(* CODESYS project CoreMotionNc2.library
   Version: 1.1.8
   Title: CoreMotionNc2
   DefaultNamespace: CoreMotionNc2
   Placeholder: CoreMotionNc2
   Company: Beckhoff Automation LLC

Project tree, tasks and I/O mapping:
  libraries: Core, * (Beckhoff Automation LLC); Tc2_MC2, * (Beckhoff Automation GmbH); Tc2_MC2_Drive, * (Beckhoff Automation GmbH); Tc2_NcKinematicTransformation, * (Beckhoff Automation GmbH); Tc2_Standard, * (Beckhoff Automation GmbH); Tc2_System, * (Beckhoff Automation GmbH)
  _Internal/
    Interface/
      interface I_AxisRef: Axis
      interface I_MotionJogTask: JogBackwards, JogForward, Mode, Position
      interface I_MotionPowerTask
      interface I_MotionTask: Axis, Name
      interface I_MotionTaskCollection: AddTask, ErrorTask, RemoveTaskByInstance
    MotionTasks/
      AX5000/
        DUT/
          P_0_0074/
            data type ST_IDN_P_0_0074
            data type ST_IDN_P_0_0074_UDINT
          P_0_0074_LREAL/
            data type ST_IDN_P_0_0074_LREAL
          data type ST_AX5000AmpToNm
        function block MotionTask_AX5000AmpToNm [ST]: ActCurrent, ActTorque, Busy, CyclicLogic, Error, ErrorId, Execute
      Base/
        DUT/
          data type ST_TaskState
        function block MotionTask [ST]: Axis, Busy, CyclicLogic, Error, ErrorId, Execute, Name
        function block MotionTaskCollection [ST]: Busy, Error, ErrorId, ErrorTask, AddTask, CyclicLogic, FB_Init, RemoveTaskByInstance, Reset
      Coupling/
        function block MotionCoupleTask_Gearing [ST]: BufferMode, Busy, CyclicLogic, Error, ErrorId, Execute, GearIn, GearInMultiMasterOptions, GearRatioMaster1, GearRatioMaster2, GearRatioMaster3, GearRatioMaster4, Master1, Master2, Master3, Master4
      Home/
        function block MotionHomeTask_CoESetEncoderOffset [ST]: Busy, CyclicLogic, Error, ErrorId, Execute, HomePosition
        function block MotionHomeTask_SetPosition [ST]: Busy, CyclicLogic, Error, ErrorId, Execute, HomePosition
        function block MotionHomeTask_SetPositionOffset [ST]: Busy, CyclicLogic, Error, ErrorId, Execute, Feedback, HomePosition, Memory
        function block MotionHomeTask_SetZeroHere [ST]: Busy, CyclicLogic, Error, ErrorId, Execute
      Move/
        function block MoveAbsoluteTask [ST]: BufferMode, Busy, CyclicLogic, Error, ErrorId, Execute, MoveOptions, TargetPosition
        function block MoveJogTask [ST]: Busy, CyclicLogic, Error, ErrorId, Execute, JogBackwards, JogForward, Mode, Position
        function block MoveModuloTask [ST]: BufferMode, Busy, CyclicLogic, Direction, Error, ErrorId, Execute, MoveOptions, TargetPosition
        function block MoveRelativeTask [ST]: BufferMode, Busy, CyclicLogic, Error, ErrorId, Execute, MoveOptions, TargetDistance
        function block MoveVelocityTask [ST]: BufferMode, Busy, CyclicLogic, Error, ErrorId, Execute, MoveOptions, TargetVelocity
      Power/
        function block PowerTask [ST]: Busy, CyclicLogic, Disable, Enable, Enabled, Error, ErrorId, Execute, InhibitFeedBackward, InhibitFeedForward, Override
        function block StopTask [ST]: BufferMode, Busy, CyclicLogic, Error, ErrorId, Execute, MoveOptions
      Reset/
        function block CoEExtendedResetTask [ST]: Busy, CyclicLogic, Error, ErrorId, Execute
        function block CoEResetTask [ST]: Busy, CyclicLogic, Error, ErrorId, Execute
        function block SoEResetTask [ST]: Busy, CyclicLogic, Error, ErrorId, Execute
  Kinematic Group/
    Interface/
      interface I_KinematicGroup: AddAcsAxis, AddMcsAxis, BuildGroup, DissolveGroup, Status
    function block KinematicGroup [ST]: DeregisterWithParent, RegisterWithParent, CyclicLogic, Initialize, Initialized, AddAcsAxis, AddMcsAxis, BuildGroup, DissolveGroup, Override, Status, Reset, Busy, Error, ErrorId
    function block KinematicGroup_TcEvents [ST]: GetHighestActiveEventReaction, GetHighestActiveEventSeverity, Reset, SetEventReactions, CyclicLogic, FB_Init
  Motion/
    DUT/
      data type ST_AxisPTP_HMI
      data type ST_MotionDefaults
    Interface/
      interface I_Axis: ErrorId, MotionTasks
      interface I_Axis_PTP
      interface I_AxisDynamics: Acceleration, BufferMode, Deceleration, Jerk, MoveOptions, Velocity
      interface I_AxisEnable: InhibitFeedBackward, InhibitFeedForward
      interface I_AxisGear: GearIn, GearInMultiMasterOptions, GearOut, GearRatioMaster1, GearRatioMaster2, GearRatioMaster3, GearRatioMaster4, Master1, Master2, Master3, Master4
      interface I_AxisHome: Home
      interface I_AxisJog: Jog
      interface I_AxisMoveAbsolute: MoveAbsolute
      interface I_AxisMoveModulo: MoveModulo
      interface I_AxisMoveRelative: MoveRelative
      interface I_AxisMoveVelocity: MoveVelocity
      interface I_AxisStatus: ActualAcceleration, ActualPosition, ActualPositionModulo, ActualTorque, ActualVelocity, AxisParameterSet, Enabled, PositionLag, SetAcceleration, SetPosition, SetPositionModulo, SetVelocity, Stopped
      interface I_SlaveAxis
    function block Axis [ST]: FB_Init, RegisterWithParent, CyclicLogic, Acceleration, BufferMode, Deceleration, Jerk, MoveOptions, Velocity, Disable, Enable, Enabled, InhibitFeedBackward, InhibitFeedForward, Override, Home, HomeTask, Initialize, Initialized, Jog, Reset, ResetTask, ActualAcceleration, ActualPosition, ActualPositionModulo, ActualTorque, ActualVelocity, AxisParameterSet, Busy, Error, ErrorId, PositionLag, SetAcceleration, SetPosition, SetPositionModulo, SetVelocity, Stop, Stopped, StopTask, Axis, MotionTasks
    function block Axis_TcEvents [ST]: GetHighestActiveEventReaction, GetHighestActiveEventSeverity, Reset, SetEventReactions, CyclicLogic, FB_Init
    function block AxisPTP [ST]: FB_Init, MoveAbsolute, MoveModulo, MoveRelative, MoveVelocity
    function block AxisPTP_HMI [ST]: DisablePermissive, EnablePermissive, HomePermissive, JogBackwardFastPermissive, JogBackwardSlowPermissive, JogForwardFastPermissive, JogForwardSlowPermissive, MoveAbsolutePermissive, MoveModuloPermissive, MoveRelativePermissive, MoveVelocityPermissive, ResetPermissive, StopPermissive, ControlObject, CyclicLogic, FB_Init
    function block SlaveAxisPTP [ST]: FB_Init, GearIn, GearInMultiMasterOptions, GearOut, GearRatioMaster1, GearRatioMaster2, GearRatioMaster3, GearRatioMaster4, Master1, Master2, Master3, Master4
  Project Information/
    function F_GetCompany [ST]
    function F_GetTitle [ST]
    function F_GetVersion [ST]
  Version/
    global variables Global_Version
  global variables CoreMotionParameterNc2
*)

// _Internal/MotionTasks/AX5000/DUT/P_0_0074/ST_IDN_P_0_0074
TYPE ST_IDN_P_0_0074 :
	STRUCT
		Iq : ARRAY[0..9] OF UDINT; // Amps ( units := A x 100 )
		M  : ARRAY[0..9] OF UDINT; // Newton Meters ( units := Nm x 100 )
	END_STRUCT
END_TYPE

// _Internal/MotionTasks/AX5000/DUT/P_0_0074/ST_IDN_P_0_0074_UDINT
TYPE ST_IDN_P_0_0074_UDINT :
	STRUCT
		Actual	 : UINT;
		_Max	 : UINT;
		Elements : ST_IDN_P_0_0074;
	END_STRUCT
END_TYPE

// _Internal/MotionTasks/AX5000/DUT/P_0_0074_LREAL/ST_IDN_P_0_0074_LREAL
TYPE ST_IDN_P_0_0074_LREAL :
	STRUCT
		Iq : ARRAY[0..9] OF LREAL;
		M  : ARRAY[0..9] OF LREAL;
	END_STRUCT
END_TYPE

// _Internal/MotionTasks/AX5000/DUT/ST_AX5000AmpToNm
TYPE ST_AX5000AmpToNm :
	STRUCT
		Curve	   : ST_IDN_P_0_0074_LREAL; // Contents read in from P-0-0074   ( scaled )
		ActCurrent : LREAL;					// Actual current in Amps           ( units := A )
		ActTorque  : LREAL;					// Actual torque in Newton Meters   ( units := Nm )
	END_STRUCT
END_TYPE

// _Internal/MotionTasks/Base/DUT/ST_TaskState
TYPE ST_TaskState :
	STRUCT
		Name	: T_MaxString;
		Busy	: BOOL;
		Error	: BOOL;
		ErrorId : UDINT;
	END_STRUCT
END_TYPE

// Motion/DUT/ST_AxisPTP_HMI
TYPE ST_AxisPTP_HMI EXTENDS ST_HmiFunction :
	STRUCT
		Unit				 : STRING;
		Busy				 : BOOL;
		Error				 : BOOL;
		ErrorId				 : UDINT;
		ActualAcceleration	 : LREAL;
		ActualPosition		 : LREAL;
		ActualPositionModulo : LREAL;
		ActualTorque		 : LREAL;
		ActualVelocity		 : LREAL;
		Status				 : ST_AxisStatus;
		Enable				 : Button;
		Disable				 : Button;
		Stop				 : Button;
		JogForwardSlow		 : Button;
		JogBackwardSlow		 : Button;
		JogForwardFast		 : Button;
		JogBackwardFast		 : Button;
		Home				 : Button;
		Reset				 : Button;
		MoveAbsolute		 : Button;
		TargetPosition		 : LREAL;
		MoveVelocity		 : Button;
		TargetVelocity		 : LREAL;
		MoveRelative		 : Button;
		TargetDistance		 : LREAL;
		MoveModulo			 : Button;
	END_STRUCT
END_TYPE

// Motion/DUT/ST_MotionDefaults
TYPE ST_MotionDefaults :
	STRUCT
		DefaultResetTask : CoEResetTask				  := (Name := 'MC Reset (CoE)');
		DefaultHomeTask	 : MotionHomeTask_SetZeroHere := (Name := 'MC Home');
		DefaultStopTask	 : StopTask					  := (Name := 'MC Stop');
	END_STRUCT
END_TYPE

// Version/Global_Version
{attribute 'TcGenerated'}
{attribute 'no-analysis'}
{attribute 'linkalways'}
// This function has been automatically generated from the project information.
VAR_GLOBAL CONSTANT
	{attribute 'const_non_replaced'}
	stLibVersion_CoreMotionNc2 : ST_LibVersion := (iMajor := 1, iMinor := 1, iBuild := 8, iRevision := 0, nFlags := 0, sVersion := '1.1.8');
END_VAR

// CoreMotionParameterNc2
{attribute 'qualified_only'}
VAR_GLOBAL CONSTANT
	MaxMotionTasks : UDINT := 10;
END_VAR

// _Internal/Interface/I_AxisRef
INTERFACE I_AxisRef

PROPERTY Axis : REFERENCE TO AXIS_REF
GET
END_GET
END_PROPERTY

END_INTERFACE

// Motion/Axis
FUNCTION_BLOCK Axis EXTENDS CyclicComponent IMPLEMENTS I_Initializable, I_Axis
VAR
	_Axis				 : REFERENCE TO AXIS_REF;
	Defaults			 : ST_MotionDefaults;
	MotionTaskCollection : MotionTaskCollection<CoreMotionParameterNc2.MaxMotionTasks>(THIS^);

	// Tasks
	{attribute 'hide'}
	PowerTask : PowerTask := (Name := 'MC Power');
	{attribute 'hide'}
	JogTask : MoveJogTask := (Name := 'MC Jog');
	{attribute 'hide'}
	_StopTask : I_MotionTask := Defaults.DefaultStopTask;
	{attribute 'hide'}
	_ResetTask : I_MotionTask := Defaults.DefaultResetTask;
	{attribute 'hide'}
	_HomeTask : I_MotionTask := Defaults.DefaultHomeTask;

	//
	{attribute 'hide'}
	MCReadParameterSet : MC_ReadParameterSet;
	_AxisParameters	   : ST_AxisParameterSet;
	{attribute 'hide'}
	_Initialized : BOOL;
	{attribute 'hide'}
	_Acceleration : LREAL;
	{attribute 'hide'}
	_Deceleration : LREAL;
	{attribute 'hide'}
	_Velocity : LREAL;
	{attribute 'hide'}
	_Jerk		  : LREAL;
	_McBufferMode : MC_BufferMode;
	_MoveOptions  : ST_MoveOptions;
END_VAR

(*FB_Init is always available implicitly and it is used primarily for initialization.
The return value is not evaluated. For a specific influence, you can also declare the
methods explicitly and provide additional code there with the standard initialization
code. You can evaluate the return value.*)
METHOD FB_Init : BOOL
VAR_INPUT
	(* TRUE: the retain variables are initialized (reset warm / reset cold)*)
	bInitRetains : BOOL;

	(* TRUE: the instance will be copied to the copy code afterward (online change)   *)
	bInCopyCode : BOOL;
	Name		: Core.T_MaxString;
	Axis		: REFERENCE TO AXIS_REF;
END_VAR
_Axis REF= Axis;

// Register all Motion Tasks to Collection
MotionTaskCollection.AddTask(PowerTask);
MotionTaskCollection.AddTask(_StopTask);
MotionTaskCollection.AddTask(_ResetTask);
MotionTaskCollection.AddTask(_HomeTask);
MotionTaskCollection.AddTask(JogTask);
END_METHOD

METHOD RegisterWithParent
VAR_INPUT
	Parent : Core.I_ContainComponents;
END_VAR
SUPER^.RegisterWithParent(Parent);
Parent.RegisterInitialize(THIS^);
END_METHOD

METHOD CyclicLogic
IF NOT _Initialized THEN
	Initialize();
	RETURN;
END_IF

_Axis.ReadStatus();
MotionTaskCollection.CyclicLogic();
END_METHOD

{attribute 'monitoring' := 'call'}
PROPERTY Acceleration : LREAL
GET
Acceleration := _Acceleration;
END_GET
SET
_Acceleration := Acceleration;
END_SET
END_PROPERTY

PROPERTY BufferMode : REFERENCE TO MC_BufferMode
GET
BufferMode REF= _McBufferMode;
END_GET
END_PROPERTY

{attribute 'monitoring' := 'call'}
PROPERTY Deceleration : LREAL
GET
Deceleration := _Deceleration;
END_GET
SET
_Deceleration := Deceleration;
END_SET
END_PROPERTY

{attribute 'monitoring' := 'call'}
PROPERTY Jerk : LREAL
GET
Jerk := _Jerk;
END_GET
SET
_Jerk := Jerk;
END_SET
END_PROPERTY

PROPERTY MoveOptions : REFERENCE TO ST_MoveOptions
GET
MoveOptions REF= _MoveOptions;
END_GET
END_PROPERTY

{attribute 'monitoring' := 'call'}
PROPERTY Velocity : LREAL
GET
Velocity := _Velocity;
END_GET
SET
_Velocity := Velocity;
END_SET
END_PROPERTY

METHOD Disable
PowerTask.Disable();
END_METHOD

METHOD Enable
IF Error THEN
	RETURN;
END_IF

PowerTask.Enable();
END_METHOD

{attribute 'monitoring' := 'call'}
PROPERTY Enabled : BOOL
GET
Enabled := PowerTask.Enabled;
END_GET
END_PROPERTY

{attribute 'monitoring' := 'call'}
PROPERTY InhibitFeedBackward : BOOL
GET
InhibitFeedBackward := PowerTask.InhibitFeedBackward;
END_GET
SET
PowerTask.InhibitFeedBackward := InhibitFeedBackward;
END_SET
END_PROPERTY

{attribute 'monitoring' := 'call'}
PROPERTY InhibitFeedForward : BOOL
GET
InhibitFeedForward := PowerTask.InhibitFeedForward;
END_GET
SET
PowerTask.InhibitFeedForward := InhibitFeedForward;
END_SET
END_PROPERTY

{attribute 'monitoring' := 'call'}
PROPERTY Override : LREAL
SET
PowerTask.Override := Override;
END_SET
END_PROPERTY

METHOD Home
VAR_INPUT
END_VAR
_HomeTask.Execute();
END_METHOD

PROPERTY HomeTask : I_MotionTask
SET
MotionTaskCollection.RemoveTaskByInstance(_HomeTask);
_HomeTask := HomeTask;
MotionTaskCollection.AddTask(_HomeTask);
END_SET
END_PROPERTY

METHOD Initialize
IF NOT _Initialized THEN
	MCReadParameterSet(Parameter := _AxisParameters, Axis := _Axis, Execute := TRUE);
	IF NOT MCReadParameterSet.Busy THEN
		IF MCReadParameterSet.Error THEN
			Trace.LogMessage(_Name, 'Axis not initialized - McReadParameter failed!');
		ELSIF MCReadParameterSet.Done THEN
			_Velocity	  := _AxisParameters.fVeloSlowManual;
			_Acceleration := _AxisParameters.fAcceleration;
			_Deceleration := _AxisParameters.fDeceleration;
			_Jerk		  := _AxisParameters.fJerk;
			Trace.LogMessage(_Name, 'Axis initialization complete');
			_Initialized := TRUE;
		END_IF

		MCReadParameterSet(Parameter := _AxisParameters, Axis := _Axis, Execute := FALSE);
	END_IF
END_IF
END_METHOD

{attribute 'monitoring' := 'call'}
PROPERTY Initialized : BOOL
GET
Initialized := _Initialized;
END_GET
SET
_Initialized := Initialized;
END_SET
END_PROPERTY

METHOD Jog
VAR_INPUT
	JogForward	 : BOOL;
	JogBackwards : BOOL;
	JogMode		 : E_JogMode := E_JogMode.MC_JOGMODE_STANDARD_SLOW;
	Position	 : LREAL	 := 0;
END_VAR
IF Error THEN
	RETURN;
END_IF

JogTask.JogBackwards := JogBackwards;
JogTask.JogForward	 := JogForward;
JogTask.Position	 := Position;
JogTask.Mode		 := JogMode;
JogTask.Execute();
END_METHOD

METHOD Reset
IF _ResetTask.Execute() THEN
	MotionTaskCollection.Reset();
END_IF
END_METHOD

PROPERTY ResetTask : I_MotionTask
SET
MotionTaskCollection.RemoveTaskByInstance(_ResetTask);
_ResetTask := ResetTask;
MotionTaskCollection.AddTask(_ResetTask);
END_SET
END_PROPERTY

{attribute 'monitoring' := 'call'}
PROPERTY ActualAcceleration : LREAL
GET
ActualAcceleration := _Axis.NcToPlc.ActAcc;
END_GET
END_PROPERTY

{attribute 'monitoring' := 'call'}
PROPERTY ActualPosition : LREAL
GET
ActualPosition := _Axis.NcToPlc.ActPos;
END_GET
END_PROPERTY

{attribute 'monitoring' := 'call'}
PROPERTY ActualPositionModulo : LREAL
GET
ActualPositionModulo := _Axis.NcToPlc.ModuloActPos;
END_GET
END_PROPERTY

{attribute 'monitoring' := 'call'}
PROPERTY ActualTorque : LREAL
GET
ActualTorque := _Axis.NcToPlc.ActTorque;
END_GET
END_PROPERTY

{attribute 'monitoring' := 'call'}
PROPERTY ActualVelocity : LREAL
GET
ActualVelocity := _Axis.NcToPlc.ActVelo;
END_GET
END_PROPERTY

PROPERTY AxisParameterSet : REFERENCE TO ST_AxisParameterSet
GET
AxisParameterSet REF= _AxisParameters;
END_GET
END_PROPERTY

{attribute 'monitoring' := 'call'}
PROPERTY Busy : BOOL
GET
Busy := MotionTaskCollection.Busy;
END_GET
END_PROPERTY

{attribute 'monitoring' := 'call'}
PROPERTY Error : BOOL
GET
Error := MotionTaskCollection.Error OR _Axis.Status.Error;
END_GET
END_PROPERTY

{attribute 'monitoring' := 'call'}
PROPERTY ErrorId : UDINT
GET
IF _Axis.Status.ErrorID <> 0 THEN
	ErrorId := _Axis.Status.ErrorID;
	RETURN;
END_IF

ErrorId := MotionTaskCollection.ErrorId;
END_GET
END_PROPERTY

{attribute 'monitoring' := 'call'}
PROPERTY PositionLag : LREAL
GET
PositionLag := _Axis.NcToPlc.PosDiff;
END_GET
END_PROPERTY

{attribute 'monitoring' := 'call'}
PROPERTY SetAcceleration : LREAL
GET
SetAcceleration := _Axis.NcToPlc.SetAcc;
END_GET
END_PROPERTY

{attribute 'monitoring' := 'call'}
PROPERTY SetPosition : LREAL
GET
SetPosition := _Axis.NcToPlc.SetPos;
END_GET
END_PROPERTY

{attribute 'monitoring' := 'call'}
PROPERTY SetPositionModulo : LREAL
GET
SetPositionModulo := _Axis.NcToPlc.ModuloSetPos;
END_GET
END_PROPERTY

{attribute 'monitoring' := 'call'}
PROPERTY SetVelocity : LREAL
GET
SetVelocity := _Axis.NcToPlc.SetVelo;
END_GET
END_PROPERTY

METHOD Stop
IF Error AND _Axis.Status.Error THEN
	(* It's possible that a function block errored but
	not the NC itself--in this case we can allow a stop command.
	If the NC Axis has a real fault then we want a successful reset first *)
	RETURN;
END_IF

_StopTask.Execute();
END_METHOD

{attribute 'monitoring' := 'call'}
PROPERTY Stopped : BOOL
GET
Stopped := _Axis.Status.NotMoving;
END_GET
END_PROPERTY

PROPERTY StopTask : I_MotionTask
SET
MotionTaskCollection.RemoveTaskByInstance(_StopTask);
_StopTask := StopTask;
MotionTaskCollection.AddTask(_ResetTask);
END_SET
END_PROPERTY

PROPERTY Axis : REFERENCE TO AXIS_REF
GET
Axis REF= _Axis;
END_GET
END_PROPERTY

PROPERTY MotionTasks : I_MotionTaskCollection
GET
MotionTasks := MotionTaskCollection;
END_GET
END_PROPERTY

END_FUNCTION_BLOCK

// Motion/Interface/I_Axis
INTERFACE I_Axis EXTENDS I_Component, I_AxisEnable, I_AxisRef, I_Resettable, I_Stoppable, I_AxisDynamics, I_AxisStatus, I_AxisJog, I_AxisHome

{attribute 'monitoring' := 'call'}
PROPERTY ErrorId : UDINT
GET
END_GET
END_PROPERTY

PROPERTY MotionTasks : I_MotionTaskCollection
GET
END_GET
END_PROPERTY

END_INTERFACE

// Motion/Interface/I_AxisEnable
INTERFACE I_AxisEnable EXTENDS I_Enablable, I_Override

{attribute 'monitoring' := 'call'}
PROPERTY InhibitFeedBackward : BOOL
GET
END_GET
SET
END_SET
END_PROPERTY

{attribute 'monitoring' := 'call'}
PROPERTY InhibitFeedForward : BOOL
GET
END_GET
SET
END_SET
END_PROPERTY

END_INTERFACE

// Motion/Interface/I_AxisDynamics
INTERFACE I_AxisDynamics EXTENDS I_Base

{attribute 'monitoring' := 'call'}
PROPERTY Acceleration : LREAL
GET
END_GET
SET
END_SET
END_PROPERTY

PROPERTY BufferMode : REFERENCE TO MC_BufferMode
GET
END_GET
END_PROPERTY

{attribute 'monitoring' := 'call'}
PROPERTY Deceleration : LREAL
GET
END_GET
SET
END_SET
END_PROPERTY

{attribute 'monitoring' := 'call'}
PROPERTY Jerk : LREAL
GET
END_GET
SET
END_SET
END_PROPERTY

PROPERTY MoveOptions : REFERENCE TO ST_MoveOptions
GET
END_GET
END_PROPERTY

{attribute 'monitoring' := 'call'}
PROPERTY Velocity : LREAL
GET
END_GET
SET
END_SET
END_PROPERTY

END_INTERFACE

// Motion/Interface/I_AxisStatus
INTERFACE I_AxisStatus EXTENDS I_Base, I_TaskResult

{attribute 'monitoring' := 'call'}
PROPERTY ActualAcceleration : LREAL
GET
END_GET
END_PROPERTY

{attribute 'monitoring' := 'call'}
PROPERTY ActualPosition : LREAL
GET
END_GET
END_PROPERTY

{attribute 'monitoring' := 'call'}
PROPERTY ActualPositionModulo : LREAL
GET
END_GET
END_PROPERTY

{attribute 'monitoring' := 'call'}
PROPERTY ActualTorque : LREAL
GET
END_GET
END_PROPERTY

{attribute 'monitoring' := 'call'}
PROPERTY ActualVelocity : LREAL
GET
END_GET
END_PROPERTY

PROPERTY AxisParameterSet : REFERENCE TO ST_AxisParameterSet
GET
END_GET
END_PROPERTY

{attribute 'monitoring' := 'call'}
PROPERTY Enabled : BOOL
GET
END_GET
END_PROPERTY

{attribute 'monitoring' := 'call'}
PROPERTY PositionLag : LREAL
GET
END_GET
END_PROPERTY

{attribute 'monitoring' := 'call'}
PROPERTY SetAcceleration : LREAL
GET
END_GET
END_PROPERTY

{attribute 'monitoring' := 'call'}
PROPERTY SetPosition : LREAL
GET
END_GET
END_PROPERTY

{attribute 'monitoring' := 'call'}
PROPERTY SetPositionModulo : LREAL
GET
END_GET
END_PROPERTY

{attribute 'monitoring' := 'call'}
PROPERTY SetVelocity : LREAL
GET
END_GET
END_PROPERTY

{attribute 'monitoring' := 'call'}
PROPERTY Stopped : BOOL
GET
END_GET
END_PROPERTY

END_INTERFACE

// Motion/Interface/I_AxisJog
INTERFACE I_AxisJog EXTENDS I_Base

METHOD Jog
VAR_INPUT
	JogForward	 : BOOL;
	JogBackwards : BOOL;
	JogMode		 : E_JogMode := E_JogMode.MC_JOGMODE_STANDARD_SLOW;
	Position	 : LREAL	 := 0;
END_VAR
END_METHOD

END_INTERFACE

// Motion/Interface/I_AxisHome
INTERFACE I_AxisHome EXTENDS I_Base

METHOD Home
VAR_INPUT
END_VAR
END_METHOD

END_INTERFACE

// _Internal/Interface/I_MotionTaskCollection
INTERFACE I_MotionTaskCollection EXTENDS I_TaskResult

METHOD AddTask
VAR_INPUT
	Task : I_MotionTask;
END_VAR
END_METHOD

{attribute 'monitoring' := 'call'}
PROPERTY ErrorTask : T_MaxString
GET
END_GET
END_PROPERTY

METHOD RemoveTaskByInstance
VAR_INPUT
	Task : I_MotionTask;
END_VAR
END_METHOD

END_INTERFACE

// _Internal/Interface/I_MotionTask
INTERFACE I_MotionTask EXTENDS I_Cyclic, I_TaskResult, I_Command

PROPERTY Axis : I_Axis
GET
END_GET
SET
END_SET
END_PROPERTY

{attribute 'monitoring' := 'call'}
PROPERTY Name : T_MaxString
GET
END_GET
SET
END_SET
END_PROPERTY

END_INTERFACE

// _Internal/MotionTasks/Base/MotionTaskCollection
FUNCTION_BLOCK MotionTaskCollection
VAR_GENERIC CONSTANT
	MaxCount : UDINT := 10;
END_VAR IMPLEMENTS I_MotionTaskCollection, I_Cyclic, I_Resettable
VAR
	MotionTasks		   : ARRAY[0..MaxCount] OF I_MotionTask;
	Axis			   : I_Axis;
	LastBusyTaskState  : ST_TaskState;
	LastErrorTaskState : ST_TaskState;
	CurrentTaskStates  : ARRAY[0..MaxCount] OF ST_TaskState;
	{attribute 'hide'}
	_Busy : BOOL;
	{attribute 'hide'}
	_Error : BOOL;
	{attribute 'hide'}
	_ErrorId : UDINT;
	{attribute 'hide'}
	_ErrorTask : T_MaxString;
END_VAR

{attribute 'monitoring' := 'call'}
PROPERTY Busy : BOOL
GET
Busy := _Busy;
END_GET
END_PROPERTY

{attribute 'monitoring' := 'call'}
PROPERTY Error : BOOL
GET
Error := _Error;
END_GET
END_PROPERTY

{attribute 'monitoring' := 'call'}
PROPERTY ErrorId : UDINT
GET
ErrorId := _ErrorId;
END_GET
END_PROPERTY

{attribute 'monitoring' := 'call'}
PROPERTY ErrorTask : T_MaxString
GET
ErrorTask := _ErrorTask;
END_GET
END_PROPERTY

METHOD AddTask
VAR_INPUT
	Task : I_MotionTask;
END_VAR

VAR
	i : UDINT;
END_VAR
Task.Axis := Axis;
FOR i := 0 TO MaxCount DO
	IF MotionTasks[i] = 0 THEN
		MotionTasks[i] := Task;
		EXIT;
	END_IF
END_FOR
END_METHOD

METHOD CyclicLogic
VAR
	MotionTask : I_MotionTask;
END_VAR

VAR_INST
	i				: UDINT;
END_VAR
_Busy := FALSE;
FOR i := 0 TO MaxCount DO
	IF MotionTasks[i] = 0 THEN
		EXIT;
	END_IF

	MotionTasks[i].CyclicLogic();
	IF MotionTasks[i].Busy THEN
		LastBusyTaskState.Name	  := MotionTasks[i].Name;
		LastBusyTaskState.Busy	  := MotionTasks[i].Busy;
		LastBusyTaskState.Error	  := MotionTasks[i].Error;
		LastBusyTaskState.ErrorId := MotionTasks[i].ErrorId;
		_Busy					  := TRUE;
	END_IF

	IF MotionTasks[i].Error AND NOT _Error THEN
		LastErrorTaskState.Name	   := MotionTasks[i].Name;
		LastErrorTaskState.Busy	   := MotionTasks[i].Busy;
		LastErrorTaskState.Error   := MotionTasks[i].Error;
		LastErrorTaskState.ErrorId := MotionTasks[i].ErrorId;
		_Error					   := TRUE;
		_ErrorId				   := MotionTasks[i].ErrorId;
		_ErrorTask				   := MotionTasks[i].Name;
	END_IF

	CurrentTaskStates[i].Name	 := MotionTasks[i].Name;
	CurrentTaskStates[i].Busy	 := MotionTasks[i].Busy;
	CurrentTaskStates[i].Error	 := MotionTasks[i].Error;
	CurrentTaskStates[i].ErrorId := MotionTasks[i].ErrorId;
END_FOR
END_METHOD

//FB_Init is always available implicitly and it is used primarily for initialization.

//The return value is not evaluated. For a specific influence, you can also declare the

//methods explicitly and provide additional code there with the standard initialization

//code. You can evaluate the return value.
METHOD FB_Init : BOOL
VAR_INPUT
	bInitRetains : BOOL; // TRUE: the retain variables are initialized (reset warm / reset cold)
	bInCopyCode	 : BOOL; // TRUE: the instance will be copied to the copy code afterward (online change)  
	Axis		 : I_Axis;
END_VAR
THIS^.Axis := Axis;
END_METHOD

METHOD RemoveTaskByInstance
VAR_INPUT
	Task : I_MotionTask;
END_VAR

VAR
	i : UDINT;
END_VAR
FOR i := 0 TO MaxCount DO
	IF MotionTasks[i] = Task THEN
		MotionTasks[i] := 0;
		EXIT;
	END_IF
END_FOR
END_METHOD

METHOD Reset
_Error	   := FALSE;
_ErrorId   := 0;
_ErrorTask := '';
END_METHOD

END_FUNCTION_BLOCK

// _Internal/MotionTasks/Base/MotionTask
FUNCTION_BLOCK ABSTRACT MotionTask IMPLEMENTS I_MotionTask
VAR
	_Name : T_MaxString;
	_Axis : I_Axis;
END_VAR

PROPERTY Axis : I_Axis
GET
Axis := _Axis;
END_GET
SET
_Axis := Axis;
END_SET
END_PROPERTY

{attribute 'monitoring' := 'call'}
PROPERTY ABSTRACT Busy : BOOL
GET
END_GET
END_PROPERTY

METHOD ABSTRACT CyclicLogic
END_METHOD

{attribute 'monitoring' := 'call'}
PROPERTY ABSTRACT Error : BOOL
GET
END_GET
END_PROPERTY

{attribute 'monitoring' := 'call'}
PROPERTY ABSTRACT ErrorId : UDINT
GET
END_GET
END_PROPERTY

METHOD ABSTRACT Execute : BOOL;
END_METHOD

{attribute 'monitoring' := 'call'}
PROPERTY Name : T_MaxString
GET
Name := _Name;
END_GET
SET
_Name := Name;
END_SET
END_PROPERTY

END_FUNCTION_BLOCK

// _Internal/MotionTasks/Power/PowerTask
FUNCTION_BLOCK PowerTask EXTENDS MotionTask IMPLEMENTS I_MotionPowerTask
VAR
	McPower : MC_Power;
	{attribute 'hide'}
	_InhibitFeedForward : BOOL;
	{attribute 'hide'}
	_InhibitFeedBackward : BOOL;
END_VAR

{attribute 'monitoring' := 'call'}
PROPERTY Busy : BOOL
GET
Busy := FALSE; (*MC Power Busy behaves busy as long as enabled*)
END_GET
END_PROPERTY

METHOD CyclicLogic
McPower(Axis := _Axis.Axis, Enable_Positive := NOT _InhibitFeedForward, Enable_Negative := NOT _InhibitFeedBackward);
END_METHOD

METHOD Disable
McPower.Enable := FALSE;
END_METHOD

METHOD Enable
McPower.Enable := TRUE;
END_METHOD

{attribute 'monitoring' := 'call'}
PROPERTY Enabled : BOOL
GET
Enabled := McPower.Status;
END_GET
END_PROPERTY

{attribute 'monitoring' := 'call'}
PROPERTY Error : BOOL
GET
Error := McPower.Error;
END_GET
END_PROPERTY

{attribute 'monitoring' := 'call'}
PROPERTY ErrorId : UDINT
GET
ErrorId := McPower.ErrorID;
END_GET
END_PROPERTY

METHOD Execute : BOOL
Execute := TRUE;
END_METHOD

{attribute 'monitoring' := 'call'}
PROPERTY InhibitFeedBackward : BOOL
GET
InhibitFeedBackward := _InhibitFeedBackward;
END_GET
SET
_InhibitFeedBackward := InhibitFeedBackward;
END_SET
END_PROPERTY

{attribute 'monitoring' := 'call'}
PROPERTY InhibitFeedForward : BOOL
GET
InhibitFeedForward := _InhibitFeedForward;
END_GET
SET
_InhibitFeedForward := InhibitFeedForward;
END_SET
END_PROPERTY

{attribute 'monitoring' := 'call'}
PROPERTY Override : LREAL
SET
McPower.Override := Override;
END_SET
END_PROPERTY

END_FUNCTION_BLOCK

// _Internal/Interface/I_MotionPowerTask
INTERFACE I_MotionPowerTask EXTENDS I_MotionTask, I_AxisEnable

END_INTERFACE

// _Internal/MotionTasks/Move/MoveJogTask
FUNCTION_BLOCK MoveJogTask EXTENDS MotionTask IMPLEMENTS I_MotionJogTask
VAR
	McJog		  : MC_Jog;
	_JogForward	  : BOOL;
	_JogBackwards : BOOL;
	_Mode		  : E_JogMode;
	_Position	  : LREAL;
END_VAR

{attribute 'monitoring' := 'call'}
PROPERTY Busy : BOOL
GET
Busy := MCJog.Busy;
END_GET
END_PROPERTY

METHOD CyclicLogic
McJog(Axis		   := _Axis.Axis,
	  Velocity	   := _Axis.Velocity,
	  Acceleration := _Axis.Acceleration,
	  Deceleration := _Axis.Deceleration,
	  Jerk		   := _Axis.Jerk);
END_METHOD

{attribute 'monitoring' := 'call'}
PROPERTY Error : BOOL
GET
Error := MCJog.Error;
END_GET
END_PROPERTY

{attribute 'monitoring' := 'call'}
PROPERTY ErrorId : UDINT
GET
ErrorId := MCJog.ErrorID;
END_GET
END_PROPERTY

METHOD Execute : BOOL
McJog(Axis		   := _Axis.Axis,
	  JogForward   := _JogForward,
	  JogBackwards := _JogBackwards,
	  Mode		   := _Mode,
	  Position	   := _Position);
END_METHOD

PROPERTY JogBackwards : BOOL
SET
_JogBackwards := JogBackwards;
END_SET
END_PROPERTY

PROPERTY JogForward : BOOL
SET
_JogForward := JogForward;
END_SET
END_PROPERTY

PROPERTY Mode : E_JogMode
SET
_Mode := Mode;
END_SET
END_PROPERTY

PROPERTY Position : LREAL
SET
_Position := Position;
END_SET
END_PROPERTY

END_FUNCTION_BLOCK

// _Internal/Interface/I_MotionJogTask
INTERFACE I_MotionJogTask EXTENDS I_MotionTask

PROPERTY JogBackwards : BOOL
SET
END_SET
END_PROPERTY

PROPERTY JogForward : BOOL
SET
END_SET
END_PROPERTY

PROPERTY Mode : E_JogMode
SET
END_SET
END_PROPERTY

PROPERTY Position : LREAL
SET
END_SET
END_PROPERTY

END_INTERFACE

// _Internal/MotionTasks/Power/StopTask
FUNCTION_BLOCK StopTask EXTENDS MotionTask IMPLEMENTS I_MotionTask
VAR
	McHalt		  : MC_Halt;
	_McBufferMode : MC_BufferMode;
	_MoveOptions  : ST_MoveOptions;
END_VAR

PROPERTY BufferMode : REFERENCE TO MC_BufferMode
GET
BufferMode REF= _McBufferMode;
END_GET
END_PROPERTY

{attribute 'monitoring' := 'call'}
PROPERTY Busy : BOOL
GET
Busy := McHalt.Busy;
END_GET
END_PROPERTY

METHOD CyclicLogic
McHalt(Axis			:= _Axis.Axis,
	   Deceleration := _Axis.Deceleration,
	   Jerk			:= _Axis.Jerk,
	   BufferMode	:= _McBufferMode,
	   Options		:= _MoveOptions);

McHalt.Execute := FALSE;
END_METHOD

{attribute 'monitoring' := 'call'}
PROPERTY Error : BOOL
GET
Error := McHalt.Error;
END_GET
END_PROPERTY

{attribute 'monitoring' := 'call'}
PROPERTY ErrorId : UDINT
GET
ErrorId := McHalt.ErrorID;
END_GET
END_PROPERTY

METHOD Execute : BOOL
McHalt(Axis			:= _Axis.Axis,
	   Execute		:= TRUE,
	   Deceleration := _Axis.Deceleration,
	   Jerk			:= _Axis.Jerk,
	   BufferMode	:= _McBufferMode,
	   Options		:= _MoveOptions);

Execute := TRUE;
END_METHOD

PROPERTY MoveOptions : REFERENCE TO ST_MoveOptions
GET
MoveOptions REF= _MoveOptions;
END_GET
END_PROPERTY

END_FUNCTION_BLOCK

// _Internal/MotionTasks/AX5000/MotionTask_AX5000AmpToNm
FUNCTION_BLOCK MotionTask_AX5000AmpToNm EXTENDS MotionTask
VAR
	i					   : INT;
	SequenceState		   : DINT := -10;
	RawConfigChPeakCurrent : UDINT;					// Configured Channel Peak Current  ( raw )
	ConfigChPeakCurrent	   : LREAL;					// Configured Channel Peak Current  ( units := A )
	MotorConsType		   : WORD;					// Motor construction type          ( raw )
	MotorType			   : BOOL;					// Motor construction type          ( units := 0 = Rotary, 1 = Linear ) 
	RawContStallTorque	   : UDINT;					// Motor continuous stall torque    ( raw )
	ContStallTorque		   : LREAL;					// Motor continuous stall torque    ( units := Nm )
	ContStallTorqueEx	   : LREAL;					// Motor continuous stall torque    ( units := Nm ) - extended slope   
	RawPeakTorque		   : UDINT;					// Motor peak torque                ( raw )
	PeakTorque			   : LREAL;					// Motor peak torque                ( units := Nm )
	RawContStallForce	   : UDINT;					// Motor continuous stall force     ( raw )
	ContStallForce		   : LREAL;					// Motor continuous stall force     ( units := N )
	ContStallForceEx	   : LREAL;					// Motor continuous stall force     ( units := N ) - extended slope
	RawPeakForce		   : UDINT;					// Motor peak force                 ( raw )
	PeakForce			   : LREAL;					// Motor peak force                 ( units := N )
	RawContStallCurrent	   : UDINT;					// Motor continuous stall current   ( raw )
	ContStallCurrent	   : LREAL;					// Motor continuous stall current   ( units := A )
	ContStallCurrentEx	   : LREAL;					// Motor continuous stall current   ( units := A ) - extended slope
	RawPeakCurrent		   : UDINT;					// Motor peak current               ( raw )
	PeakCurrent			   : LREAL;					// Motor peak current               ( units := A )
	Scale				   : LREAL;					// Position between array indexes   ( units := % )
	SoERead				   : FB_SoERead;			// Read SoE params from drive
	RawMotorTorqueCurve	   : ST_IDN_P_0_0074_UDINT; // Contents read in from P-0-0074   ( raw )
END_VAR

VAR
	_ErrorId		 : UDINT;			 // 1 = Axis Not Linked, 2 = Failed To Read P-0-0074, 3 = Failed To Read P-0-0092, 4 = Failed To Read P-0-0050, 5 = Failed To Read P-0-0070, 6 = Failed To Read P-0-0126, 7 = Failed To Read S-0-0111
	CalculatedValues : ST_AX5000AmpToNm; // Data read in and calculated from the drive
END_VAR

(*  
Error Ids:
  1 = Axis Not Linked, 
  2 = Failed To Read P-0-0074,
  3 = Failed To Read P-0-0092, 
  4 = Failed To Read P-0-0050, 
  5 = Failed To Read P-0-0070, 
  6 = Failed To Read P-0-0126, 
  7 = Failed To Read S-0-0111 
*)

{attribute 'monitoring' := 'call'}
PROPERTY ActCurrent : LREAL
GET
ActCurrent := CalculatedValues.ActCurrent;
END_GET
END_PROPERTY

{attribute 'monitoring' := 'call'}
PROPERTY ActTorque : LREAL
GET
ActTorque := CalculatedValues.ActTorque;
END_GET
END_PROPERTY

{attribute 'monitoring' := 'call'}
PROPERTY Busy : BOOL
GET
Busy := SequenceState > 0 AND SequenceState <= 100;
END_GET
END_PROPERTY

METHOD CyclicLogic
IF _Axis = 0 THEN
	RETURN;
END_IF

CASE SequenceState OF
	-10: // Initialize
		RawConfigChPeakCurrent := 0;
		ConfigChPeakCurrent	   := 0.0;
		MotorConsType		   := 0;
		MotorType			   := FALSE;
		RawContStallTorque	   := 0;
		ContStallTorque		   := 0.0;
		ContStallTorqueEx	   := 0.0;
		RawPeakTorque		   := 0;
		PeakTorque			   := 0.0;
		RawContStallForce	   := 0;
		ContStallForce		   := 0.0;
		ContStallForceEx	   := 0.0;
		RawPeakForce		   := 0;
		PeakForce			   := 0.0;
		RawContStallCurrent	   := 0;
		ContStallCurrent	   := 0.0;
		ContStallCurrentEx	   := 0.0;
		RawPeakCurrent		   := 0;
		PeakCurrent			   := 0.0;
		Scale				   := 0.0;
		SoERead(Execute := FALSE, Axis := _Axis.Axis);
		MEMSET(ADR(RawMotorTorqueCurve), 16#0, SIZEOF(RawMotorTorqueCurve));
		MEMSET(ADR(CalculatedValues), 16#0, SIZEOF(CalculatedValues));
		IF _Axis.Axis.NcToPlc.AxisId = 0 THEN
			_ErrorId	  := 1;
			SequenceState := 5000;
		ELSE
			SequenceState := SequenceState + 10;
		END_IF

	0:	// Wait for Execute()  
	10: // Read in the value of P-0-0074 ( Motor torque characteristic )
		SoERead(NetId	:= '',
				Idn		:= P_0_IDNs + 74,
				Element := 16#40,
				pDstBuf := ADR(RawMotorTorqueCurve),
				BufLen	:= SIZEOF(RawMotorTorqueCurve),
				Execute := TRUE,
				Axis	:= _Axis.Axis);

		IF NOT SoERead.Busy AND NOT SoERead.Error THEN
			SoERead(Execute := FALSE, Axis := _Axis.Axis);
			FOR i := 0 TO 9 DO // Convert raw values into actual units
				CalculatedValues.Curve.Iq[i] := UDINT_TO_LREAL(RawMotorTorqueCurve.Elements.Iq[i]) / 1000.0;
				CalculatedValues.Curve.M[i]	 := UDINT_TO_LREAL(RawMotorTorqueCurve.Elements.M[i]) / 100.0;
			END_FOR

			SequenceState := SequenceState + 10;
		ELSIF SoERead.Error THEN
			SoERead(Execute := FALSE, Axis := _Axis.Axis);
			_ErrorId	  := 2;
			SequenceState := 5000;
		END_IF

	20: // Read in the value of P-0-0092 ( Configured channel peak current )       
		SoERead(NetId	:= '',
				Idn		:= P_0_IDNs + 92,
				Element := 16#40,
				pDstBuf := ADR(RawConfigChPeakCurrent),
				BufLen	:= SIZEOF(RawConfigChPeakCurrent),
				Execute := TRUE,
				Axis	:= _Axis.Axis);

		IF NOT SoERead.Busy AND NOT SoERead.Error THEN // Convert raw values into actual units
			SoERead(Execute := FALSE, Axis := _Axis.Axis);
			ConfigChPeakCurrent := UDINT_TO_LREAL(RawConfigChPeakCurrent) / 1000.0;
			SequenceState		:= SequenceState + 10;
		ELSIF SoERead.Error THEN
			SoERead(Execute := FALSE, Axis := _Axis.Axis);
			_ErrorId	  := 3;
			SequenceState := 5000;
		END_IF

	30: // Check for valid characteristic curve
		IF RawMotorTorqueCurve.Elements.Iq[9] = 0 THEN
			SequenceState := SequenceState + 10; // Curve is not available
		ELSE
			SequenceState := 1000; // Curve is available
		END_IF

	40: // Read in the value of P-0-0050 ( Motor construction type )       
		SoERead(NetId	:= '',
				Idn		:= P_0_IDNs + 50,
				Element := 16#40,
				pDstBuf := ADR(MotorConsType),
				BufLen	:= SIZEOF(MotorConsType),
				Execute := TRUE,
				Axis	:= _Axis.Axis);

		IF NOT SoERead.Busy AND NOT SoERead.Error THEN
			SoERead(Execute := FALSE, Axis := _Axis.Axis);
			MotorType := MotorConsType.1;
			IF NOT MotorType THEN
				SequenceState := 50; // Rotary
			ELSE
				SequenceState := 70; // Linear
			END_IF
		ELSIF SoERead.Error THEN
			SoERead(Execute := FALSE, Axis := _Axis.Axis);
			_ErrorId	  := 4;
			SequenceState := 5000;
		END_IF

	50: // Read in the value of P-0-0070 ( Motor continuous stall torque )       
		SoERead(NetId	:= '',
				Idn		:= P_0_IDNs + 70,
				Element := 16#40,
				pDstBuf := ADR(RawContStallTorque),
				BufLen	:= SIZEOF(RawContStallTorque),
				Execute := TRUE,
				Axis	:= _Axis.Axis);

		IF NOT SoERead.Busy AND NOT SoERead.Error THEN
			SoERead(Execute := FALSE, Axis := _Axis.Axis);
			ContStallTorque := UDINT_TO_LREAL(RawContStallTorque) / 100.0;
			SequenceState	:= SequenceState + 10;
		ELSIF SoERead.Error THEN
			SoERead(Execute := FALSE, Axis := _Axis.Axis);
			_ErrorId	  := 5;
			SequenceState := 5000;
		END_IF

	60: // Read in the value of P-0-0073 ( Motor peak torque )       
		SoERead(NetId	:= '',
				Idn		:= P_0_IDNs + 73,
				Element := 16#40,
				pDstBuf := ADR(RawPeakTorque),
				BufLen	:= SIZEOF(RawPeakTorque),
				Execute := TRUE,
				Axis	:= _Axis.Axis);

		IF NOT SoERead.Busy AND NOT SoERead.Error THEN
			SoERead(Execute := FALSE, Axis := _Axis.Axis);
			PeakTorque	  := UDINT_TO_LREAL(RawPeakTorque) / 100.0;
			SequenceState := 90;
		ELSIF SoERead.Error THEN
			SoERead(Execute := FALSE, Axis := _Axis.Axis);
			SequenceState := 90;
		END_IF

	70: // Read in the value of P-0-0126 ( Motor continuous stall force )       
		SoERead(NetId	:= '',
				Idn		:= P_0_IDNs + 126,
				Element := 16#40,
				pDstBuf := ADR(RawContStallForce),
				BufLen	:= SIZEOF(RawContStallForce),
				Execute := TRUE,
				Axis	:= _Axis.Axis);

		IF NOT SoERead.Busy AND NOT SoERead.Error THEN
			SoERead(Execute := FALSE, Axis := _Axis.Axis);
			ContStallForce := UDINT_TO_LREAL(RawContStallForce) / 100.0;
			SequenceState  := SequenceState + 10;
		ELSIF SoERead.Error THEN
			SoERead(Execute := FALSE, Axis := _Axis.Axis);
			_ErrorId	  := 6;
			SequenceState := 5000;
		END_IF

	80: // Read in the value of P-0-0128 ( Motor peak force )       
		SoERead(NetId	:= '',
				Idn		:= P_0_IDNs + 128,
				Element := 16#40,
				pDstBuf := ADR(RawPeakForce),
				BufLen	:= SIZEOF(RawPeakForce),
				Execute := TRUE,
				Axis	:= _Axis.Axis);

		IF NOT SoERead.Busy AND NOT SoERead.Error THEN
			SoERead(Execute := FALSE, Axis := _Axis.Axis);
			PeakForce	  := UDINT_TO_LREAL(RawPeakForce) / 100.0;
			SequenceState := SequenceState + 10;
		ELSIF SoERead.Error THEN
			SoERead(Execute := FALSE, Axis := _Axis.Axis);
			SequenceState := SequenceState + 10;
		END_IF

	90: // Read in the value of S-0-0111 ( Motor continuous stall current )       
		SoERead(NetId	:= '',
				Idn		:= S_0_IDNs + 111,
				Element := 16#40,
				pDstBuf := ADR(RawContStallCurrent),
				BufLen	:= SIZEOF(RawContStallCurrent),
				Execute := TRUE,
				Axis	:= _Axis.Axis);

		IF NOT SoERead.Busy AND NOT SoERead.Error THEN
			SoERead(Execute := FALSE, Axis := _Axis.Axis);
			ContStallCurrent := UDINT_TO_LREAL(RawContStallCurrent) / 1000.0;
			SequenceState	 := SequenceState + 10;
		ELSIF SoERead.Error THEN
			SoERead(Execute := FALSE, Axis := _Axis.Axis);
			_ErrorId	  := 7;
			SequenceState := 5000;
		END_IF

	100: // Read in the value of S-0-0109 ( Motor peak current )       
		SoERead(NetId	:= '',
				Idn		:= S_0_IDNs + 109,
				Element := 16#40,
				pDstBuf := ADR(RawPeakCurrent),
				BufLen	:= SIZEOF(RawPeakCurrent),
				Execute := TRUE,
				Axis	:= _Axis.Axis);

		IF NOT SoERead.Busy THEN
			SoERead(Execute := FALSE, Axis := _Axis.Axis);
			PeakCurrent := UDINT_TO_LREAL(RawPeakCurrent) / 1000.0;
			IF NOT MotorType THEN
				IF PeakCurrent = 0 OR PeakTorque = 0 THEN
					SequenceState := 300; // Rotary Motor: Curve not available... peak torque and current missing - Using slope of points 0,0 to P-0-0070 and S-0-0111
				ELSE
					SequenceState := 200; // Rotary Motor: Curve not available - Using linear interpolation of points P-0-0070, P-0-0073, S-0-0111 and S-0-0109
				END_IF
			ELSE
				IF PeakCurrent = 0 OR PeakForce = 0 THEN
					SequenceState := 500; // Linear Motor: Curve not available... peak torque and current missing - Using slope of points 0,0 to P-0-0126 and S-0-0111
				ELSE
					SequenceState := 400; // Linear Motor: Curve not available - Using linear interpolation of points P-0-0126, P-0-0128, S-0-0111 and S-0-0109
				END_IF
			END_IF
		END_IF

	200: // Rotary Motor: Curve not available - Using linear interpolation of points P-0-0070, P-0-0073, S-0-0111 and S-0-0109
		CalculatedValues.ActCurrent := ABS((_Axis.Axis.NcToPlc.ActTorque / 100) * ConfigChPeakCurrent);
		// Convert the actual current in amps to Nm
		IF CalculatedValues.ActCurrent = 0 THEN
			CalculatedValues.ActTorque := 0;
		ELSIF CalculatedValues.ActCurrent > 0 AND CalculatedValues.ActCurrent < ContStallCurrent THEN
			IF ContStallCurrent > 0 THEN
				Scale					   := CalculatedValues.ActCurrent / ContStallCurrent;
				CalculatedValues.ActTorque := Scale * ContStallTorque;
			END_IF
		ELSIF CalculatedValues.ActCurrent >= ContStallCurrent AND CalculatedValues.ActCurrent <= PeakCurrent THEN
			IF (CalculatedValues.ActCurrent - ContStallCurrent) > 0 AND (PeakCurrent - ContStallCurrent) > 0 THEN
				Scale					   := (CalculatedValues.ActCurrent - ContStallCurrent) / (PeakCurrent - ContStallCurrent);
				CalculatedValues.ActTorque := (Scale * (PeakTorque - ContStallTorque) + ContStallTorque);
			END_IF
		END_IF

	300: // Rotary Motor: Curve not available... peak torque and current missing - Using slope of points 0,0 to P-0-0070 and S-0-0111
		CalculatedValues.ActCurrent := ABS((_Axis.Axis.NcToPlc.ActTorque / 100) * ConfigChPeakCurrent);

		// Project slope from continuous stall torque/current
		ContStallCurrentEx := ContStallCurrent * 10.0;
		ContStallTorqueEx  := ContStallTorque * 10.0;
		// Convert the actual current in amps to Nm
		IF CalculatedValues.ActCurrent = 0 THEN
			CalculatedValues.ActTorque := 0;
		ELSIF CalculatedValues.ActCurrent > 0 AND CalculatedValues.ActCurrent <= ContStallCurrentEx THEN
			IF ContStallCurrentEx > 0 THEN
				Scale					   := CalculatedValues.ActCurrent / ContStallCurrentEx;
				CalculatedValues.ActTorque := Scale * ContStallTorqueEx;
			END_IF
		END_IF

	400: // Linear Motor: Curve not available - Using linear interpolation of points P-0-0126, P-0-0128, S-0-0111 and S-0-0109
		CalculatedValues.ActCurrent := ABS((_Axis.Axis.NcToPlc.ActTorque / 100) * ConfigChPeakCurrent);
		// Convert the actual current in amps to Nm
		IF CalculatedValues.ActCurrent = 0 THEN
			CalculatedValues.ActTorque := 0;
		ELSIF CalculatedValues.ActCurrent > 0 AND CalculatedValues.ActCurrent < ContStallCurrent THEN
			IF ContStallCurrent > 0 THEN
				Scale					   := CalculatedValues.ActCurrent / ContStallCurrent;
				CalculatedValues.ActTorque := Scale * ContStallForce;
			END_IF
		ELSIF CalculatedValues.ActCurrent >= ContStallCurrent AND CalculatedValues.ActCurrent <= PeakCurrent THEN
			IF (CalculatedValues.ActCurrent - ContStallCurrent) > 0 AND (PeakCurrent - ContStallCurrent) > 0 THEN
				Scale					   := (CalculatedValues.ActCurrent - ContStallCurrent) / (PeakCurrent - ContStallCurrent);
				CalculatedValues.ActTorque := (Scale * (PeakForce - ContStallForce) + ContStallForce);
			END_IF
		END_IF

	500: // Linear Motor: Curve not available... peak torque and current missing - Using slope of points 0,0 to P-0-0126 and S-0-0111
		CalculatedValues.ActCurrent := ABS((_Axis.Axis.NcToPlc.ActTorque / 100) * ConfigChPeakCurrent);

		// Project slope from continuous stall torque/current
		ContStallCurrentEx := ContStallCurrent * 10.0;
		ContStallForceEx   := ContStallForce * 10.0;
		// Convert the actual current in amps to Nm
		IF CalculatedValues.ActCurrent = 0 THEN
			CalculatedValues.ActTorque := 0;
		ELSIF CalculatedValues.ActCurrent > 0 AND CalculatedValues.ActCurrent <= ContStallCurrentEx THEN
			IF ContStallCurrentEx > 0 THEN
				Scale					   := CalculatedValues.ActCurrent / ContStallCurrentEx;
				CalculatedValues.ActTorque := Scale * ContStallForceEx;
			END_IF
		END_IF

	1000: // Rotary or Linear Motor: Curve available - Compare actual torque value in Amps to the characteristic curve and output actual torque value in Nm
		CalculatedValues.ActCurrent := ABS((_Axis.Axis.NcToPlc.ActTorque / 100) * ConfigChPeakCurrent);
		// Convert the actual current in amps to Nm
		FOR i := 1 TO 9 DO
			IF CalculatedValues.ActCurrent = 0 THEN
				CalculatedValues.ActTorque := 0;
				EXIT;
			ELSIF CalculatedValues.ActCurrent > 0 AND CalculatedValues.ActCurrent < CalculatedValues.Curve.Iq[0] THEN
				IF CalculatedValues.Curve.Iq[0] > 0 THEN
					Scale					   := CalculatedValues.ActCurrent / CalculatedValues.Curve.Iq[0];
					CalculatedValues.ActTorque := Scale * CalculatedValues.Curve.M[0];
				END_IF

				EXIT;
			ELSIF CalculatedValues.ActCurrent >= CalculatedValues.Curve.Iq[i - 1] AND CalculatedValues.ActCurrent <= CalculatedValues.Curve.Iq[i] THEN
				IF (CalculatedValues.Curve.Iq[i] - CalculatedValues.Curve.Iq[i - 1]) > 0 AND CalculatedValues.ActCurrent - CalculatedValues.Curve.Iq[i - 1] > 0 THEN
					Scale					   := (CalculatedValues.ActCurrent - CalculatedValues.Curve.Iq[i - 1]) / (CalculatedValues.Curve.Iq[i] - CalculatedValues.Curve.Iq[i - 1]);
					CalculatedValues.ActTorque := (Scale * (CalculatedValues.Curve.M[i] - CalculatedValues.Curve.M[i - 1]) + CalculatedValues.Curve.M[i - 1]);
				END_IF

				EXIT;
			END_IF
		END_FOR

	5000: // Error state        
		SequenceState := -10;
END_CASE
END_METHOD

{attribute 'monitoring' := 'call'}
PROPERTY Error : BOOL
GET
Error := SequenceState = 5000;
END_GET
END_PROPERTY

{attribute 'monitoring' := 'call'}
PROPERTY ErrorId : UDINT
GET
ErrorId := _ErrorId;
END_GET
END_PROPERTY

METHOD Execute : BOOL
IF Busy THEN
	RETURN;
END_IF

SequenceState := 10;
_ErrorID	  := 0;
Execute		  := TRUE;
END_METHOD

END_FUNCTION_BLOCK

// _Internal/MotionTasks/Coupling/MotionCoupleTask_Gearing
FUNCTION_BLOCK MotionCoupleTask_Gearing EXTENDS MotionTask
VAR
	McGearInMultimaster : MC_GearInMultiMaster;
	McGearOut			: MC_GearOut;
	{attribute 'hide'}
	_GearIn : BOOL;
	{attribute 'hide'}
	_GearRatioMaster1 : LREAL := 1.0;
	{attribute 'hide'}
	_GearRatioMaster2 : LREAL := 1.0;
	{attribute 'hide'}
	_GearRatioMaster3 : LREAL := 1.0;
	{attribute 'hide'}
	_GearRatioMaster4 : LREAL := 1.0;
	{attribute 'hide'}
	DummyAxis : AXIS_REF;
	{attribute 'hide'}
	MasterAxis1 : REFERENCE TO AXIS_REF;
	{attribute 'hide'}
	MasterAxis2 : REFERENCE TO AXIS_REF;
	{attribute 'hide'}
	MasterAxis3 : REFERENCE TO AXIS_REF;
	{attribute 'hide'}
	MasterAxis4				  : REFERENCE TO AXIS_REF;
	_Master1				  : I_Axis;
	_Master2				  : I_Axis;
	_Master3				  : I_Axis;
	_Master4				  : I_Axis;
	_McBufferMode			  : MC_BufferMode;
	_GearInMultiMasterOptions : ST_GearInMultiMasterOptions;
END_VAR

PROPERTY BufferMode : MC_BufferMode
SET
_McBufferMode := BufferMode;
END_SET
END_PROPERTY

{attribute 'monitoring' := 'call'}
PROPERTY Busy : BOOL
GET
END_GET
END_PROPERTY

METHOD CyclicLogic
IF _Master1 <> 0 THEN
	MasterAxis1 REF= _Master1.Axis;
ELSE
	MasterAxis1 REF= DummyAxis;
END_IF

IF _Master2 <> 0 THEN
	MasterAxis2 REF= _Master2.Axis;
ELSE
	MasterAxis2 REF= DummyAxis;
END_IF

IF _Master3 <> 0 THEN
	MasterAxis3 REF= _Master3.Axis;
ELSE
	MasterAxis3 REF= DummyAxis;
END_IF

IF _Master4 <> 0 THEN
	MasterAxis4 REF= _Master4.Axis;
ELSE
	MasterAxis4 REF= DummyAxis;
END_IF

McGearInMultimaster(Master1		 := MasterAxis1,
					Master2		 := MasterAxis2,
					Master3		 := MasterAxis3,
					Master4		 := MasterAxis4,
					Slave		 := _Axis.Axis,
					GearRatio1	 := _GearRatioMaster1,
					GearRatio2	 := _GearRatioMaster2,
					GearRatio3	 := _GearRatioMaster3,
					GearRatio4	 := _GearRatioMaster4,
					Acceleration := _Axis.Acceleration,
					Deceleration := _Axis.Deceleration,
					Jerk		 := _Axis.Jerk,
					BufferMode	 := _McBufferMode,
					Options		 :=);

McGearOut(Slave := _Axis.Axis);
McGearOut.Execute := FALSE;
END_METHOD

{attribute 'monitoring' := 'call'}
PROPERTY Error : BOOL
GET
Error := McGearInMultimaster.Error;
END_GET
END_PROPERTY

{attribute 'monitoring' := 'call'}
PROPERTY ErrorId : UDINT
GET
ErrorId := McGearInMultimaster.ErrorID;
END_GET
END_PROPERTY

METHOD Execute : BOOL
IF _GearIn THEN
	IF _Axis.Error OR Busy THEN
		RETURN;
	END_IF

	McGearInMultimaster.Enable := TRUE;
ELSE
	IF Busy THEN
		RETURN;
	END_IF

	McGearOut.Execute		   := TRUE;
	McGearInMultimaster.Enable := FALSE;
END_IF

Execute := TRUE;
END_METHOD

PROPERTY GearIn : BOOL
SET
_GearIn := GearIn;
END_SET
END_PROPERTY

PROPERTY GearInMultiMasterOptions : ST_GearInMultiMasterOptions
SET
_GearInMultiMasterOptions := GearInMultiMasterOptions;
END_SET
END_PROPERTY

{attribute 'monitoring' := 'call'}
PROPERTY GearRatioMaster1 : LREAL
SET
_GearRatioMaster1 := GearRatioMaster1;
END_SET
END_PROPERTY

{attribute 'monitoring' := 'call'}
PROPERTY GearRatioMaster2 : LREAL
SET
_GearRatioMaster2 := GearRatioMaster2;
END_SET
END_PROPERTY

{attribute 'monitoring' := 'call'}
PROPERTY GearRatioMaster3 : LREAL
SET
_GearRatioMaster3 := GearRatioMaster3;
END_SET
END_PROPERTY

{attribute 'monitoring' := 'call'}
PROPERTY GearRatioMaster4 : LREAL
SET
_GearRatioMaster4 := GearRatioMaster4;
END_SET
END_PROPERTY

PROPERTY Master1 : I_Axis
SET
_Master1 := Master1;
END_SET
END_PROPERTY

PROPERTY Master2 : I_Axis
SET
_Master2 := Master2;
END_SET
END_PROPERTY

PROPERTY Master3 : I_Axis
SET
_Master3 := Master3;
END_SET
END_PROPERTY

PROPERTY Master4 : I_Axis
SET
_Master4 := Master4;
END_SET
END_PROPERTY

END_FUNCTION_BLOCK

// _Internal/MotionTasks/Home/MotionHomeTask_CoESetEncoderOffset
FUNCTION_BLOCK MotionHomeTask_CoESetEncoderOffset EXTENDS MotionTask
VAR
	SequenceState	  : UDINT;
	SetPositionOffset : FB_CoEAX8000SetPositionOffset;
	_HomePosition	  : LREAL := 0.0;
	_ErrorId		  : UDINT;
END_VAR

{attribute 'monitoring' := 'call'}
PROPERTY Busy : BOOL
GET
Busy := SequenceState <> 0;
END_GET
END_PROPERTY

METHOD CyclicLogic
VAR_INST
	DriveEnabledAtBeginning : BOOL;
	AxisRef					: REFERENCE TO AXIS_REF;
END_VAR
CASE SequenceState OF
	0: // Wait for Execute();
	10:
		IF Axis.Enabled THEN
			DriveEnabledAtBeginning := TRUE;
			SequenceState			:= 20;
		ELSE
			DriveEnabledAtBeginning := FALSE;
			SequenceState			:= 30;
		END_IF

	20:
		Axis.Disable();
		IF NOT Axis.Enabled THEN
			SequenceState := 30;
		END_IF

	30:
		AxisRef REF= Axis.Axis;
		SetPositionOffset(Axis	   := AxisRef,
						  Execute  := TRUE,
						  Position := _HomePosition,
						  Relative := FALSE,
						  Feedback := ePositionOffsetFeedback1,
						  Memory   := ePositionOffsetMemory_Encoder);

		IF NOT SetPositionOffset.Busy THEN
			IF SetPositionOffset.Error THEN
				_ErrorId	  := SetPositionOffset.ErrorID;
				SequenceState := 999;
			ELSE
				SequenceState := 40;
			END_IF

			SetPositionOffset(Axis := AxisRef, Execute := FALSE);
		END_IF

	40:
		IF DriveEnabledAtBeginning THEN
			SequenceState := 50;
		ELSE
			SequenceState := 0;
		END_IF

	50:
		Axis.Enable();
		IF Axis.Enabled THEN
			SequenceState := 0;
		END_IF

	999:
		_ErrorId	  := 0;
		SequenceState := 0;
END_CASE
END_METHOD

{attribute 'monitoring' := 'call'}
PROPERTY Error : BOOL
GET
Error := SequenceState = 999;
END_GET
END_PROPERTY

{attribute 'monitoring' := 'call'}
PROPERTY ErrorId : UDINT
GET
ErrorId := _ErrorId;
END_GET
END_PROPERTY

METHOD Execute : BOOL
IF Axis.Busy OR Axis.Error THEN
	RETURN;
END_IF

SequenceState := 10;
_ErrorID	  := 0;
Execute		  := TRUE;
END_METHOD

{attribute 'monitoring' := 'call'}
PROPERTY HomePosition : LREAL
GET
HomePosition := _HomePosition;
END_GET
SET
_HomePosition := HomePosition;
END_SET
END_PROPERTY

END_FUNCTION_BLOCK

// _Internal/MotionTasks/Home/MotionHomeTask_SetPosition
FUNCTION_BLOCK MotionHomeTask_SetPosition EXTENDS MotionTask
VAR
	MCSetPosition : MC_SetPosition;
	_HomePosition : LREAL := 0.0;
END_VAR

{attribute 'monitoring' := 'call'}
PROPERTY Busy : BOOL
GET
Busy := MCSetPosition.Busy;
END_GET
END_PROPERTY

METHOD CyclicLogic
MCSetPosition(Axis := _Axis.Axis, Position := HomePosition);
MCSetPosition.Execute := FALSE;
END_METHOD

{attribute 'monitoring' := 'call'}
PROPERTY Error : BOOL
GET
Error := MCSetPosition.Error;
END_GET
END_PROPERTY

{attribute 'monitoring' := 'call'}
PROPERTY ErrorId : UDINT
GET
ErrorId := MCSetPosition.ErrorID;
END_GET
END_PROPERTY

METHOD Execute : BOOL
IF Axis.Busy OR Axis.Error THEN
	RETURN;
END_IF

MCSetPosition.Execute := TRUE;
Execute				  := TRUE;
END_METHOD

PROPERTY HomePosition : LREAL
GET
HomePosition := MCSetPosition.Position;
END_GET
SET
MCSetPosition.Position := HomePosition;
END_SET
END_PROPERTY

END_FUNCTION_BLOCK

// _Internal/MotionTasks/Home/MotionHomeTask_SetPositionOffset
FUNCTION_BLOCK MotionHomeTask_SetPositionOffset EXTENDS MotionTask
VAR
	SequenceState	  : UDINT;
	SetPositionOffset : FB_SetPositionOffset;
	_HomePosition	  : LREAL := 0.0;
	_ErrorId		  : UDINT;
	_Feedback		  : E_PositionOffsetFeedback := E_PositionOffsetFeedback.ePositionOffsetFeedback1;
	_Memory			  : E_PositionOffsetMemory	 := E_PositionOffsetMemory.ePositionOffsetMemory_Encoder;
END_VAR

{attribute 'monitoring' := 'call'}
PROPERTY Busy : BOOL
GET
Busy := SequenceState <> 0;
END_GET
END_PROPERTY

METHOD CyclicLogic
VAR_INST
	DriveEnabledAtBeginning : BOOL;
	AxisRef					: REFERENCE TO AXIS_REF;
END_VAR
CASE SequenceState OF
	0: // Wait for Execute();
	10:
		IF Axis.Enabled THEN
			DriveEnabledAtBeginning := TRUE;
			SequenceState			:= 20;
		ELSE
			DriveEnabledAtBeginning := FALSE;
			SequenceState			:= 30;
		END_IF

	20:
		Axis.Disable();
		IF NOT Axis.Enabled THEN
			SequenceState := 30;
		END_IF

	30:
		AxisRef REF= Axis.Axis;
		SetPositionOffset(Axis	   := AxisRef,
						  Execute  := TRUE,
						  Position := _HomePosition,
						  Relative := FALSE,
						  Feedback := _Feedback,
						  Memory   := _Memory);

		IF NOT SetPositionOffset.Busy THEN
			IF SetPositionOffset.Error THEN
				_ErrorId	  := SetPositionOffset.ErrorID;
				SequenceState := 999;
			ELSE
				SequenceState := 40;
			END_IF

			SetPositionOffset(Axis := AxisRef, Execute := FALSE);
		END_IF

	40:
		IF DriveEnabledAtBeginning THEN
			SequenceState := 50;
		ELSE
			SequenceState := 0;
		END_IF

	50:
		Axis.Enable();
		IF Axis.Enabled THEN
			SequenceState := 0;
		END_IF

	999:
		_ErrorId	  := 0;
		SequenceState := 0;
END_CASE
END_METHOD

{attribute 'monitoring' := 'call'}
PROPERTY Error : BOOL
GET
Error := SequenceState = 999;
END_GET
END_PROPERTY

{attribute 'monitoring' := 'call'}
PROPERTY ErrorId : UDINT
GET
ErrorId := _ErrorId;
END_GET
END_PROPERTY

METHOD Execute : BOOL
IF Axis.Busy OR Axis.Error THEN
	RETURN;
END_IF

SequenceState := 10;
_ErrorID	  := 0;
Execute		  := TRUE;
END_METHOD

{attribute 'monitoring' := 'call'}
PROPERTY Feedback : E_PositionOffsetFeedback
SET
_Feedback := Feedback;
END_SET
END_PROPERTY

{attribute 'monitoring' := 'call'}
PROPERTY HomePosition : LREAL
GET
HomePosition := _HomePosition;
END_GET
SET
_HomePosition := HomePosition;
END_SET
END_PROPERTY

{attribute 'monitoring' := 'call'}
PROPERTY Memory : E_PositionOffsetMemory
SET
_Memory := Memory;
END_SET
END_PROPERTY

END_FUNCTION_BLOCK

// _Internal/MotionTasks/Home/MotionHomeTask_SetZeroHere
FUNCTION_BLOCK MotionHomeTask_SetZeroHere EXTENDS MotionTask
VAR
	MCSetPosition : MC_SetPosition;
END_VAR

{attribute 'monitoring' := 'call'}
PROPERTY Busy : BOOL
GET
Busy := MCSetPosition.Busy;
END_GET
END_PROPERTY

METHOD CyclicLogic
MCSetPosition(Axis := _Axis.Axis);
MCSetPosition.Execute := FALSE;
END_METHOD

{attribute 'monitoring' := 'call'}
PROPERTY Error : BOOL
GET
Error := MCSetPosition.Error;
END_GET
END_PROPERTY

{attribute 'monitoring' := 'call'}
PROPERTY ErrorId : UDINT
GET
ErrorId := MCSetPosition.ErrorID;
END_GET
END_PROPERTY

METHOD Execute : BOOL
IF Axis.Busy OR Axis.Error THEN
	RETURN;
END_IF

MCSetPosition.Execute := TRUE;
Execute				  := TRUE;
END_METHOD

END_FUNCTION_BLOCK

// _Internal/MotionTasks/Move/MoveAbsoluteTask
FUNCTION_BLOCK MoveAbsoluteTask EXTENDS MotionTask
VAR
	_TargetPosition : LREAL;
	McMoveAbsolute	: ARRAY[0..1] OF MC_MoveAbsolute;
	Active			: UDINT;
	_McBufferMode	: MC_BufferMode;
	_MoveOptions	: ST_MoveOptions;
END_VAR

PROPERTY BufferMode : REFERENCE TO MC_BufferMode
GET
BufferMode REF= _McBufferMode;
END_GET
END_PROPERTY

{attribute 'monitoring' := 'call'}
PROPERTY Busy : BOOL
GET
Busy := McMoveAbsolute[Active].Busy;
END_GET
END_PROPERTY

METHOD CyclicLogic
McMoveAbsolute[Active](Axis			:= _Axis.Axis,
					   Position		:= _TargetPosition,
					   Velocity		:= _Axis.Velocity,
					   Acceleration := _Axis.Acceleration,
					   Deceleration := _Axis.Deceleration,
					   Jerk			:= _Axis.Jerk,
					   BufferMode	:= _McBufferMode,
					   Options		:= _MoveOptions);

McMoveAbsolute[Active].Execute := FALSE;
END_METHOD

{attribute 'monitoring' := 'call'}
PROPERTY Error : BOOL
GET
Error := McMoveAbsolute[Active].Error;
END_GET
END_PROPERTY

{attribute 'monitoring' := 'call'}
PROPERTY ErrorId : UDINT
GET
ErrorID := McMoveAbsolute[Active].ErrorID;
END_GET
END_PROPERTY

METHOD Execute : BOOL;
IF Active = 0 THEN
	Active := 1;
	McMoveAbsolute[Active](Axis			:= _Axis.Axis,
						   Execute		:= TRUE,
						   Position		:= _TargetPosition,
						   Velocity		:= _Axis.Velocity,
						   Acceleration := _Axis.Acceleration,
						   Deceleration := _Axis.Deceleration,
						   Jerk			:= _Axis.Jerk,
						   BufferMode	:= _McBufferMode,
						   Options		:= _MoveOptions);
ELSE
	Active := 0;
	McMoveAbsolute[Active](Axis			:= _Axis.Axis,
						   Execute		:= TRUE,
						   Position		:= _TargetPosition,
						   Velocity		:= _Axis.Velocity,
						   Acceleration := _Axis.Acceleration,
						   Deceleration := _Axis.Deceleration,
						   Jerk			:= _Axis.Jerk,
						   BufferMode	:= _McBufferMode,
						   Options		:= _MoveOptions);
END_IF

Execute := TRUE;
END_METHOD

PROPERTY MoveOptions : REFERENCE TO ST_MoveOptions
GET
MoveOptions REF= _MoveOptions;
END_GET
END_PROPERTY

{attribute 'monitoring' := 'call'}
PROPERTY TargetPosition : LREAL
SET
_TargetPosition := TargetPosition;
END_SET
END_PROPERTY

END_FUNCTION_BLOCK

// _Internal/MotionTasks/Move/MoveModuloTask
FUNCTION_BLOCK MoveModuloTask EXTENDS MotionTask
VAR
	_TargetPosition : LREAL;
	_Direction		: MC_Direction;
	McMoveModulo	: ARRAY[0..1] OF MC_MoveModulo;
	Active			: UDINT;
    _McBufferMode	: MC_BufferMode;
	_MoveOptions	: ST_MoveOptions;
END_VAR

PROPERTY BufferMode : REFERENCE TO MC_BufferMode
GET
BufferMode REF= _McBufferMode;
END_GET
END_PROPERTY

{attribute 'monitoring' := 'call'}
PROPERTY Busy : BOOL
GET
Busy := McMoveModulo[Active].Busy;
END_GET
END_PROPERTY

METHOD CyclicLogic
McMoveModulo[Active](Axis		  := _Axis.Axis,
					 Position	  := _TargetPosition,
					 Direction	  := _Direction,
					 Velocity	  := _Axis.Velocity,
					 Acceleration := _Axis.Acceleration,
					 Deceleration := _Axis.Deceleration,
					 Jerk		  := _Axis.Jerk,
					 BufferMode	  := _McBufferMode,
					 Options	  := _MoveOptions);

McMoveModulo[Active].Execute := FALSE;
END_METHOD

PROPERTY Direction : MC_Direction
SET
_Direction := Direction;
END_SET
END_PROPERTY

{attribute 'monitoring' := 'call'}
PROPERTY Error : BOOL
GET
Error := McMoveModulo[Active].Error;
END_GET
END_PROPERTY

{attribute 'monitoring' := 'call'}
PROPERTY ErrorId : UDINT
GET
ErrorID := McMoveModulo[Active].ErrorID;
END_GET
END_PROPERTY

METHOD Execute : BOOL;
IF Active = 0 THEN
	Active := 1;
	McMoveModulo[Active](Axis		  := _Axis.Axis,
						 Execute	  := TRUE,
						 Position	  := _TargetPosition,
						 Direction	  := _Direction,
						 Velocity	  := _Axis.Velocity,
						 Acceleration := _Axis.Acceleration,
						 Deceleration := _Axis.Deceleration,
						 Jerk		  := _Axis.Jerk,
						 BufferMode	  := _McBufferMode,
						 Options	  := _MoveOptions);
ELSE
	Active := 0;
	McMoveModulo[Active](Axis		  := _Axis.Axis,
						 Execute	  := TRUE,
						 Position	  := _TargetPosition,
						 Direction	  := _Direction,
						 Velocity	  := _Axis.Velocity,
						 Acceleration := _Axis.Acceleration,
						 Deceleration := _Axis.Deceleration,
						 Jerk		  := _Axis.Jerk,
						 BufferMode	  := _McBufferMode,
						 Options	  := _MoveOptions);
END_IF

Execute := TRUE;
END_METHOD

PROPERTY MoveOptions : REFERENCE TO ST_MoveOptions
GET
MoveOptions REF= _MoveOptions;
END_GET
END_PROPERTY

{attribute 'monitoring' := 'call'}
PROPERTY TargetPosition : LREAL
SET
_TargetPosition := TargetPosition;
END_SET
END_PROPERTY

END_FUNCTION_BLOCK

// _Internal/MotionTasks/Move/MoveRelativeTask
FUNCTION_BLOCK MoveRelativeTask EXTENDS MotionTask
VAR
	_TargetDistance : LREAL;
	McMoveRelative	: ARRAY[0..1] OF MC_MoveRelative;
	Active			: UDINT;
    _McBufferMode	: MC_BufferMode;
	_MoveOptions	: ST_MoveOptions;
END_VAR

PROPERTY BufferMode : REFERENCE TO MC_BufferMode
GET
BufferMode REF= _McBufferMode;
END_GET
END_PROPERTY

{attribute 'monitoring' := 'call'}
PROPERTY Busy : BOOL
GET
Busy := McMoveRelative[Active].Busy;
END_GET
END_PROPERTY

METHOD CyclicLogic
McMoveRelative[Active](Axis			:= _Axis.Axis,
					   Distance		:= _TargetDistance,
					   Velocity		:= _Axis.Velocity,
					   Acceleration := _Axis.Acceleration,
					   Deceleration := _Axis.Deceleration,
					   Jerk			:= _Axis.Jerk,
					   BufferMode	:= _McBufferMode,
					   Options		:= _MoveOptions);

McMoveRelative[Active].Execute := FALSE;
END_METHOD

{attribute 'monitoring' := 'call'}
PROPERTY Error : BOOL
GET
Error := McMoveRelative[Active].Error;
END_GET
END_PROPERTY

{attribute 'monitoring' := 'call'}
PROPERTY ErrorId : UDINT
GET
ErrorID := McMoveRelative[Active].ErrorID;
END_GET
END_PROPERTY

METHOD Execute : BOOL;
IF Active = 0 THEN
	Active := 1;
	McMoveRelative[Active](Axis			:= _Axis.Axis,
						   Execute		:= TRUE,
						   Distance		:= _TargetDistance,
						   Velocity		:= _Axis.Velocity,
						   Acceleration := _Axis.Acceleration,
						   Deceleration := _Axis.Deceleration,
						   Jerk			:= _Axis.Jerk,
						   BufferMode	:= _McBufferMode,
						   Options		:= _MoveOptions);
ELSE
	Active := 0;
	McMoveRelative[Active](Axis			:= _Axis.Axis,
						   Execute		:= TRUE,
						   Distance		:= _TargetDistance,
						   Velocity		:= _Axis.Velocity,
						   Acceleration := _Axis.Acceleration,
						   Deceleration := _Axis.Deceleration,
						   Jerk			:= _Axis.Jerk,
						   BufferMode	:= _McBufferMode,
						   Options		:= _MoveOptions);
END_IF

Execute := TRUE;
END_METHOD

PROPERTY MoveOptions : REFERENCE TO ST_MoveOptions
GET
MoveOptions REF= _MoveOptions;
END_GET
END_PROPERTY

{attribute 'monitoring' := 'call'}
PROPERTY TargetDistance : LREAL
SET
_TargetDistance := TargetDistance;
END_SET
END_PROPERTY

END_FUNCTION_BLOCK

// _Internal/MotionTasks/Move/MoveVelocityTask
FUNCTION_BLOCK MoveVelocityTask EXTENDS MotionTask
VAR
	_TargetVelocity : LREAL;
	McMoveVelocity	: ARRAY[0..1] OF MC_MoveVelocity;
	Active			: UDINT;
	_McBufferMode	: MC_BufferMode;
	_MoveOptions	: ST_MoveOptions;
END_VAR

PROPERTY BufferMode : REFERENCE TO MC_BufferMode
GET
BufferMode REF= _McBufferMode;
END_GET
END_PROPERTY

{attribute 'monitoring' := 'call'}
PROPERTY Busy : BOOL
GET
Busy := McMoveVelocity[Active].Busy;
END_GET
END_PROPERTY

METHOD CyclicLogic
McMoveVelocity[Active](Axis			:= _Axis.Axis,
					   Velocity		:= _TargetVelocity,
					   Acceleration := _Axis.Acceleration,
					   Deceleration := _Axis.Deceleration,
					   Jerk			:= _Axis.Jerk,
					   BufferMode	:= _McBufferMode,
					   Options		:= _MoveOptions);

McMoveVelocity[Active].Execute := FALSE;
END_METHOD

{attribute 'monitoring' := 'call'}
PROPERTY Error : BOOL
GET
Error := McMoveVelocity[Active].Error;
END_GET
END_PROPERTY

{attribute 'monitoring' := 'call'}
PROPERTY ErrorId : UDINT
GET
ErrorID := McMoveVelocity[Active].ErrorID;
END_GET
END_PROPERTY

METHOD Execute : BOOL;
IF _TargetVelocity < 0 THEN
	McMoveVelocity[Active].Direction := MC_Negative_Direction;
ELSE
	McMoveVelocity[Active].Direction := MC_Positive_Direction;
END_IF

_TargetVelocity := ABS(_TargetVelocity);
IF Active = 0 THEN
	Active := 1;
	McMoveVelocity[Active](Axis			:= _Axis.Axis,
						   Execute		:= TRUE,
						   Velocity		:= _TargetVelocity,
						   Acceleration := _Axis.Acceleration,
						   Deceleration := _Axis.Deceleration,
						   Jerk			:= _Axis.Jerk,
						   BufferMode	:= _McBufferMode,
						   Options		:= _MoveOptions);
ELSE
	Active := 0;
	McMoveVelocity[Active](Axis			:= _Axis.Axis,
						   Execute		:= TRUE,
						   Velocity		:= _TargetVelocity,
						   Acceleration := _Axis.Acceleration,
						   Deceleration := _Axis.Deceleration,
						   Jerk			:= _Axis.Jerk,
						   BufferMode	:= _McBufferMode,
						   Options		:= _MoveOptions);
END_IF

Execute := TRUE;
END_METHOD

PROPERTY MoveOptions : REFERENCE TO ST_MoveOptions
GET
MoveOptions REF= _MoveOptions;
END_GET
END_PROPERTY

{attribute 'monitoring' := 'call'}
PROPERTY TargetVelocity : LREAL
SET
_TargetVelocity := TargetVelocity;
END_SET
END_PROPERTY

END_FUNCTION_BLOCK

// _Internal/MotionTasks/Reset/CoEExtendedResetTask
FUNCTION_BLOCK CoEExtendedResetTask EXTENDS MotionTask
VAR
	DriveErrorCode AT %I* : UINT;
	CoERead				  : FB_CoERead;
	CoEWrite			  : FB_CoEWrite;
	MCReset				  : MC_Reset;
	SequenceState		  : UDINT;
	_ErrorID			  : UDINT;
END_VAR

{attribute 'monitoring' := 'call'}
PROPERTY Busy : BOOL
GET
Busy := SequenceState <> 0;
END_GET
END_PROPERTY

METHOD CyclicLogic
VAR_INST
	AlwaysTrue			 : USINT := 1;
	ExtendedResetEnabled : BOOL;
END_VAR
CASE SequenceState OF
	0: // Wait for Execute()
	10:
		IF (_Axis.Axis.Status.DriveDeviceError) THEN
			IF NOT ExtendedResetEnabled THEN
				IF (DriveErrorCode = 16#8185) OR (DriveErrorCode = 16#63A0) THEN
					SequenceState := SequenceState + 10;
				ELSIF (DriveErrorCode = 16#63A2) OR (DriveErrorCode = 16#63A4) THEN
					SequenceState := 100;
				END_IF
			ELSE
				SequenceState := 100;
			END_IF
		ELSE
			ExtendedResetEnabled := FALSE;
		END_IF

	20:
		CoEWrite(Axis	  := _Axis.Axis,
				 Index	  := 16#3004,
				 SubIndex := 16#4,
				 pSrcBuf  := ADR(AlwaysTrue),
				 BufLen	  := SIZEOF(USINT),
				 Execute  := TRUE);

		IF NOT CoEWrite.Busy THEN
			IF CoEWrite.Error THEN
				IF CoEWrite.AdsErrId > 0 THEN
					_ErrorID := CoEWrite.AdsErrId;
				ELSE
					_ErrorID := CoEWrite.CANopenErrId;
				END_IF

				SequenceState := 999;
			ELSE
				SequenceState := SequenceState + 1;
			END_IF

			CoEWrite(Axis := _Axis.Axis, Execute := FALSE);
		END_IF

	21:
		CoEWrite(Axis	  := _Axis.Axis,
				 Index	  := 16#3404,
				 SubIndex := 16#4,
				 pSrcBuf  := ADR(AlwaysTrue),
				 BufLen	  := SIZEOF(USINT),
				 Execute  := TRUE);

		IF NOT CoEWrite.Busy THEN
			IF CoEWrite.Error THEN
				IF CoEWrite.AdsErrId > 0 THEN
					_ErrorID := CoEWrite.AdsErrId;
				ELSE
					_ErrorID := CoEWrite.CANopenErrId;
				END_IF

				SequenceState := 999;
			ELSE
				SequenceState := SequenceState + 1;
			END_IF

			CoEWrite(Axis := _Axis.Axis, Execute := FALSE);
		END_IF

	22:
		ExtendedResetEnabled := TRUE;
		SequenceState		 := 1000;

	100:
		MCReset.Execute := TRUE;
		SequenceState	:= SequenceState + 10;

	110:
		IF NOT MCReset.Busy THEN
			SequenceState := 0;
		END_IF

	999:
		_ErrorID	  := 0;
		SequenceState := 0;
END_CASE

MCReset(Axis := _Axis.Axis);
MCReset.Execute := FALSE;
END_METHOD

{attribute 'monitoring' := 'call'}
PROPERTY Error : BOOL
GET
Error := SequenceState = 999;
END_GET
END_PROPERTY

{attribute 'monitoring' := 'call'}
PROPERTY ErrorId : UDINT
GET
ErrorId := _ErrorID;
END_GET
END_PROPERTY

METHOD Execute : BOOL
IF _Axis.Axis.Status.Coupled AND NOT _Axis.Axis.Status.Error THEN
	Execute := TRUE;
	RETURN;
ELSIF Busy OR _Axis.Axis.Status.Coupled THEN
	Execute := TRUE;
	RETURN;
END_IF

SequenceState := 10;
Execute		  := TRUE;
END_METHOD

END_FUNCTION_BLOCK

// _Internal/MotionTasks/Reset/CoEResetTask
FUNCTION_BLOCK CoEResetTask EXTENDS MotionTask
VAR
	MCReset		  : MC_Reset;
	SequenceState : UDINT;
END_VAR

{attribute 'monitoring' := 'call'}
PROPERTY Busy : BOOL
GET
Busy := SequenceState <> 0;
END_GET
END_PROPERTY

METHOD CyclicLogic
CASE SequenceState OF
	0: // Wait for Execute()
	10:
		MCReset.Execute := TRUE;
		SequenceState	:= SequenceState + 10;

	20:
		IF NOT MCReset.Busy THEN
			SequenceState := 0;
		END_IF
END_CASE

MCReset(Axis := _Axis.Axis);
MCReset.Execute := FALSE;
END_METHOD

{attribute 'monitoring' := 'call'}
PROPERTY Error : BOOL
GET
Error := MCReset.Error;
END_GET
END_PROPERTY

{attribute 'monitoring' := 'call'}
PROPERTY ErrorId : UDINT
GET
ErrorId := MCReset.ErrorID;
END_GET
END_PROPERTY

METHOD Execute : BOOL
IF _Axis.Axis.Status.Coupled AND NOT _Axis.Axis.Status.Error THEN
	Execute := TRUE;
	RETURN;
ELSIF Busy OR _Axis.Axis.Status.Coupled THEN
	Execute := TRUE;
	RETURN;
END_IF

SequenceState := 10;
Execute		  := TRUE;
END_METHOD

END_FUNCTION_BLOCK

// _Internal/MotionTasks/Reset/SoEResetTask
FUNCTION_BLOCK SoEResetTask EXTENDS MotionTask
VAR
	MCReset		  : MC_Reset;
	SoEReset	  : FB_SoEReset;
	SequenceState : UDINT;
	_ErrorId	  : UDINT;
END_VAR

{attribute 'monitoring' := 'call'}
PROPERTY Busy : BOOL
GET
Busy := SequenceState <> 0;
END_GET
END_PROPERTY

METHOD CyclicLogic
VAR_INST
	ResetDelay : TON;
END_VAR
CASE SequenceState OF
	0: // Wait for Execute()
	10:
		SoEReset.Execute := TRUE;
		SequenceState	 := SequenceState + 10;

	20:
		IF NOT SoEReset.Busy THEN
			IF SoEReset.Error THEN
				IF SoEReset.SercosErrId < 0 THEN
					_ErrorID := SoEReset.SercosErrId;
				ELSE
					_ErrorID := SoEReset.AdsErrId;
				END_IF

				SequenceState := 999;
			ELSE
				//No error occurred
				SequenceState := SequenceState + 10;
			END_IF
		END_IF

	30:
		MCReset.Execute := TRUE;
		SequenceState	:= SequenceState + 10;

	40:
		IF NOT MCReset.Busy THEN
			SequenceState := SequenceState + 10;
		END_IF

	50:
		ResetDelay(IN := TRUE);
		IF ResetDelay.Q OR NOT _Axis.Axis.Status.DriveDeviceError THEN
			ResetDelay(IN := FALSE);
			SequenceState := 0;
		END_IF

	999:
		_ErrorId	  := 0;
		SequenceState := 0;
END_CASE

SoEReset(Axis := _Axis.Axis);
MCReset(Axis := _Axis.Axis);
SoEReset.Execute := FALSE;
MCReset.Execute	 := FALSE;
END_METHOD

{attribute 'monitoring' := 'call'}
PROPERTY Error : BOOL
GET
Error := SequenceState = 999;
END_GET
END_PROPERTY

{attribute 'monitoring' := 'call'}
PROPERTY ErrorId : UDINT
GET
ErrorId := _ErrorID;
END_GET
END_PROPERTY

METHOD Execute : BOOL
IF _Axis.Axis.Status.Coupled AND NOT _Axis.Axis.Status.Error THEN
	Execute := TRUE;
	RETURN;
ELSIF Busy OR _Axis.Axis.Status.Coupled THEN
	Execute := TRUE;
	RETURN;
END_IF

SequenceState := 10;
Execute		  := TRUE;
END_METHOD

END_FUNCTION_BLOCK

// Kinematic Group/Interface/I_KinematicGroup
INTERFACE I_KinematicGroup EXTENDS I_Component, I_Override, I_TaskResult, I_Resettable

METHOD AddAcsAxis : BOOL
VAR_INPUT
	AxisId : UDINT;
END_VAR
END_METHOD

METHOD AddMcsAxis : BOOL
VAR_INPUT
	AxisId : UDINT;
END_VAR
END_METHOD

METHOD BuildGroup
VAR_INPUT
END_VAR
END_METHOD

METHOD DissolveGroup
VAR_INPUT
END_VAR
END_METHOD

{attribute 'monitoring' := 'call'}
PROPERTY Status : E_KinStatus
GET
END_GET
END_PROPERTY

END_INTERFACE

// Kinematic Group/KinematicGroup
FUNCTION_BLOCK KinematicGroup EXTENDS CyclicComponent IMPLEMENTS I_KinematicGroup, I_Initializable
VAR
	NcToPlc AT %I* : NCTOPLC_NCICHANNEL_REF;
	PlcToNc AT %Q* : PLCTONC_NCICHANNEL_REF;
	KinAxes		   : ST_KinAxes;
	KinConfigGroup : FB_KinConfigGroup;
	KinResetGroup  : FB_KinResetGroup;
	{attribute 'hide'}
	_Initialized : BOOL;
	{attribute 'hide'}
	_Busy : BOOL;
	{attribute 'hide'}
	_Error : BOOL;
	{attribute 'hide'}
	_ErrorId : UDINT;
END_VAR

METHOD DeregisterWithParent
VAR_INPUT
	Parent : Core.I_ContainComponents;
END_VAR
SUPER^.DeregisterWithParent(Parent);
Parent.DeregisterInitialize(THIS^);
END_METHOD

METHOD RegisterWithParent
VAR_INPUT
	Parent : Core.I_ContainComponents;
END_VAR
SUPER^.RegisterWithParent(Parent);
Parent.RegisterInitialize(THIS^);
END_METHOD

METHOD CyclicLogic
IF NOT Initialized THEN
	Initialize();
	RETURN;
END_IF

//
KinConfigGroup(stAxesList := KinAxes, stKinRefIn := NcToPlc);
IF KinConfigGroup.bError THEN
	_Error	 := TRUE;
	_ErrorId := KinConfigGroup.nErrorId;
END_IF

KinConfigGroup.bExecute := FALSE;

//
KinResetGroup(nItpChannelId := NcToPlc.ChnId, stKinRefIn := NcToPlc, stAxesList := KinAxes);
IF KinResetGroup.bError THEN
	_Error	 := TRUE;
	_ErrorId := KinResetGroup.nErrorId;
END_IF

KinResetGroup.bExecute := FALSE;

//
_Busy := KinConfigGroup.bBusy;
END_METHOD

METHOD Initialize
VAR
	i : DINT;
END_VAR
IF NOT Initialized THEN
	IF KinAxes.nAxisIdsAcs[1] = 0 THEN
		Trace.LogMessage(Name, 'Init failed - at least one ACS Axis needs to be added to Kinematic!');
		RETURN;
	END_IF

	IF KinAxes.nAxisIdsMcs[1] = 0 THEN
		Trace.LogMessage(Name, 'Init failed - at least one MCS Axis needs to be added to Kinematic!');
		RETURN;
	END_IF

	IF F_GetMappingStatus(ADR(NcToPlc), SIZEOF(NcToPlc)) <> EPlcMappingStatus.MS_Mapped THEN
		Trace.LogMessage(Name, 'Init failed - NcToPlc not mapped to Kinematic Channel!');
		RETURN;
	END_IF

	IF F_GetMappingStatus(ADR(PlcToNc), SIZEOF(PlcToNc)) <> EPlcMappingStatus.MS_Mapped THEN
		Trace.LogMessage(Name, 'Init failed - PlcToNc not mapped to Kinematic Channel!');
		RETURN;
	END_IF

	Initialized := TRUE;
END_IF
END_METHOD

{attribute 'monitoring' := 'call'}
PROPERTY Initialized : BOOL
GET
Initialized := _Initialized;
END_GET
SET
_Initialized := Initialized;
END_SET
END_PROPERTY

METHOD AddAcsAxis : BOOL
VAR_INPUT
	AxisId : UDINT;
END_VAR

VAR
	i : DINT;
END_VAR
IF AxisId = 0 THEN
	RETURN;
END_IF

FOR i := 1 TO 8 DO
	IF KinAxes.nAxisIdsAcs[i] = 0 THEN
		KinAxes.nAxisIdsAcs[i] := AxisId;
		AddAcsAxis			   := TRUE;
		RETURN;
	END_IF
END_FOR
END_METHOD

METHOD AddMcsAxis : BOOL
VAR_INPUT
	AxisId : UDINT;
END_VAR

VAR
	i : DINT;
END_VAR
IF AxisId = 0 THEN
	RETURN;
END_IF

FOR i := 1 TO 8 DO
	IF KinAxes.nAxisIdsMcs[i] = 0 THEN
		KinAxes.nAxisIdsMcs[i] := AxisId;
		AddMcsAxis			   := TRUE;
		RETURN;
	END_IF
END_FOR
END_METHOD

METHOD BuildGroup
VAR_INPUT
END_VAR
IF Busy THEN
	RETURN;
END_IF

KinConfigGroup.bCartesianMode := TRUE;
KinConfigGroup.bExecute		  := TRUE;
END_METHOD

METHOD DissolveGroup
VAR_INPUT
END_VAR
IF Busy THEN
	RETURN;
END_IF

KinConfigGroup.bCartesianMode := FALSE;
KinConfigGroup.bExecute		  := TRUE;
END_METHOD

{attribute 'monitoring' := 'call'}
PROPERTY Override : LREAL
SET
PlcToNc.ChnAxesOvr	  := TO_UDINT(Override * 10_000);
PlcToNc.ChnSpindleOvr := TO_UDINT(Override * 10_000);
END_SET
END_PROPERTY

{attribute 'monitoring' := 'call'}
PROPERTY Status : E_KinStatus
GET
Status := F_KinGetChnOperationState(NcToPlc);
END_GET
END_PROPERTY

METHOD Reset
_Error				   := FALSE;
_ErrorId			   := 0;
KinResetGroup.bExecute := TRUE;
END_METHOD

{attribute 'monitoring' := 'call'}
PROPERTY Busy : BOOL
GET
Busy := _Busy;
END_GET
END_PROPERTY

{attribute 'monitoring' := 'call'}
PROPERTY Error : BOOL
GET
Error := _Error;
END_GET
END_PROPERTY

{attribute 'monitoring' := 'call'}
PROPERTY ErrorId : UDINT
GET
ErrorId := _ErrorId;
END_GET
END_PROPERTY

END_FUNCTION_BLOCK

// Kinematic Group/KinematicGroup_TcEvents
FUNCTION_BLOCK KinematicGroup_TcEvents EXTENDS CyclicComponent IMPLEMENTS I_EventReactionTcEvents
VAR
	KinematicGroup : I_KinematicGroup;
	Events		   : TcEventClass('Kinematic Group Events');
END_VAR

METHOD GetHighestActiveEventReaction : DINT
GetHighestActiveEventReaction := Events.GetHighestActiveEventReaction();
END_METHOD

METHOD GetHighestActiveEventSeverity : Core.TcEventSeverity
GetHighestActiveEventSeverity := Events.GetHighestActiveEventSeverity();
END_METHOD

METHOD Reset
Events.Reset();
END_METHOD

METHOD SetEventReactions
VAR_INPUT
	Verbose	 : DINT := 0;
	Info	 : DINT := 1;
	Warning	 : DINT := 2;
	Error	 : DINT := 3;
	Critical : DINT := 4;
END_VAR
Events.SetEventReactions(Verbose,
						 Info,
						 Warning,
						 Error,
						 Critical);
END_METHOD

METHOD CyclicLogic
IF KinematicGroup = 0 THEN
	RETURN;
END_IF

IF KinematicGroup.Error THEN
	Events.Arguments(E_KinematicGroup.KinematicGroupError).Clear().AddString(TO_STRING(KinematicGroup.ErrorId));
	Events.RaiseEvent(E_KinematicGroup.KinematicGroupError);
END_IF
END_METHOD

(*FB_Init is always available implicitly and it is used primarily for initialization.
The return value is not evaluated. For a specific influence, you can also declare the
methods explicitly and provide additional code there with the standard initialization
code. You can evaluate the return value.*)
METHOD FB_Init : BOOL
VAR_INPUT
	(* TRUE: the retain variables are initialized (reset warm / reset cold)*)
	bInitRetains : BOOL;

	(* TRUE: the instance will be copied to the copy code afterward (online change)   *)
	bInCopyCode	   : BOOL;
	Name		   : Core.T_MaxString;
	KinematicGroup : I_KinematicGroup;
END_VAR
THIS^.KinematicGroup := KinematicGroup;
Events.GenerateTcEvents(KinematicGroup.Name, ADR(TC_Events.KinematicGroup), SIZEOF(ST_KinematicGroup));
END_METHOD

END_FUNCTION_BLOCK

// Motion/Interface/I_Axis_PTP
INTERFACE I_Axis_PTP EXTENDS I_Axis, I_AxisMoveAbsolute, I_AxisMoveModulo, I_AxisMoveRelative, I_AxisMoveVelocity

END_INTERFACE

// Motion/Interface/I_AxisMoveAbsolute
INTERFACE I_AxisMoveAbsolute EXTENDS I_Base

METHOD MoveAbsolute
VAR_INPUT
	TargetPosition : LREAL;
	AbortPrevious  : BOOL := TRUE;
END_VAR
END_METHOD

END_INTERFACE

// Motion/Interface/I_AxisMoveModulo
INTERFACE I_AxisMoveModulo EXTENDS I_Base

METHOD MoveModulo : BOOL
VAR_INPUT
	Position	  : LREAL;
	Direction	  : MC_Direction := MC_Direction.MC_Shortest_Way;
	AbortPrevious : BOOL		 := TRUE;
END_VAR
END_METHOD

END_INTERFACE

// Motion/Interface/I_AxisMoveRelative
INTERFACE I_AxisMoveRelative EXTENDS I_Base

METHOD MoveRelative : BOOL
VAR_INPUT
	Distance	  : LREAL;
	AbortPrevious : BOOL := TRUE;
END_VAR
END_METHOD

END_INTERFACE

// Motion/Interface/I_AxisMoveVelocity
INTERFACE I_AxisMoveVelocity EXTENDS I_Base

METHOD MoveVelocity : BOOL
VAR_INPUT
	Velocity	  : LREAL;
	AbortPrevious : BOOL := TRUE;
END_VAR
END_METHOD

END_INTERFACE

// Motion/Interface/I_AxisGear
INTERFACE I_AxisGear EXTENDS I_Base

METHOD GearIn
VAR_INPUT
END_VAR
END_METHOD

PROPERTY GearInMultiMasterOptions : ST_GearInMultiMasterOptions
SET
END_SET
END_PROPERTY

METHOD GearOut
VAR_INPUT
END_VAR
END_METHOD

{attribute 'monitoring' := 'call'}
PROPERTY GearRatioMaster1 : LREAL
SET
END_SET
END_PROPERTY

{attribute 'monitoring' := 'call'}
PROPERTY GearRatioMaster2 : LREAL
SET
END_SET
END_PROPERTY

{attribute 'monitoring' := 'call'}
PROPERTY GearRatioMaster3 : LREAL
SET
END_SET
END_PROPERTY

{attribute 'monitoring' := 'call'}
PROPERTY GearRatioMaster4 : LREAL
SET
END_SET
END_PROPERTY

PROPERTY Master1 : I_Axis
SET
END_SET
END_PROPERTY

PROPERTY Master2 : I_Axis
SET
END_SET
END_PROPERTY

PROPERTY Master3 : I_Axis
SET
END_SET
END_PROPERTY

PROPERTY Master4 : I_Axis
SET
END_SET
END_PROPERTY

END_INTERFACE

// Motion/Interface/I_SlaveAxis
INTERFACE I_SlaveAxis EXTENDS I_Axis_PTP, I_AxisGear

END_INTERFACE

// Motion/Axis_TcEvents
FUNCTION_BLOCK Axis_TcEvents EXTENDS CyclicComponent IMPLEMENTS I_EventReactionTcEvents
VAR
	Axis   : I_Axis;
	Events : TcEventClass(CONCAT(Name, ' Events'));
END_VAR

METHOD GetHighestActiveEventReaction : DINT
GetHighestActiveEventReaction := Events.GetHighestActiveEventReaction();
END_METHOD

METHOD GetHighestActiveEventSeverity : Core.TcEventSeverity
GetHighestActiveEventSeverity := Events.GetHighestActiveEventSeverity();
END_METHOD

METHOD Reset
Events.Reset();
END_METHOD

METHOD SetEventReactions
VAR_INPUT
	Verbose	 : DINT := 0;
	Info	 : DINT := 1;
	Warning	 : DINT := 2;
	Error	 : DINT := 3;
	Critical : DINT := 4;
END_VAR
Events.SetEventReactions(Verbose,
						 Info,
						 Warning,
						 Error,
						 Critical);
END_METHOD

METHOD CyclicLogic
IF Axis.MotionTasks.Error THEN
	Events.Arguments(E_Nc2Axis.AxisError).Clear().AddString(Axis.MotionTasks.ErrorTask).AddString(TO_STRING(Axis.MotionTasks.ErrorId));
	Events.RaiseEvent(E_Nc2Axis.AxisError);
END_IF
END_METHOD

(*FB_Init is always available implicitly and it is used primarily for initialization.
The return value is not evaluated. For a specific influence, you can also declare the
methods explicitly and provide additional code there with the standard initialization
code. You can evaluate the return value.*)
METHOD FB_Init : BOOL
VAR_INPUT
	(* TRUE: the retain variables are initialized (reset warm / reset cold)*)
	bInitRetains : BOOL;

	(* TRUE: the instance will be copied to the copy code afterward (online change)   *)
	bInCopyCode : BOOL;
	Name		: Core.T_MaxString;
	Axis		: I_Axis;
END_VAR
THIS^.Axis := Axis;
Events.GenerateTcEvents(Axis.Name, ADR(TC_events.Nc2Axis), SIZEOF(ST_Nc2Axis));
END_METHOD

END_FUNCTION_BLOCK

// Motion/AxisPTP
FUNCTION_BLOCK AxisPTP EXTENDS Axis IMPLEMENTS I_Axis_PTP
VAR
	// Tasks
	{attribute 'hide'}
	MoveAbsoluteTask : MoveAbsoluteTask := (Name := 'MC Move Absolute');
	{attribute 'hide'}
	MoveRelativeTask : MoveRelativeTask := (Name := 'MC Move Relative');
	{attribute 'hide'}
	MoveModuloTask : MoveModuloTask := (Name := 'MC Move Modulo');
	{attribute 'hide'}
	MoveVelocityTask : MoveVelocityTask := (Name := 'MC Move Velocity');
END_VAR

(*FB_Init is always available implicitly and it is used primarily for initialization.
The return value is not evaluated. For a specific influence, you can also declare the
methods explicitly and provide additional code there with the standard initialization
code. You can evaluate the return value.*)
METHOD FB_Init : BOOL
VAR_INPUT
	(* TRUE: the retain variables are initialized (reset warm / reset cold)*)
	bInitRetains : BOOL;

	(* TRUE: the instance will be copied to the copy code afterward (online change)   *)
	bInCopyCode : BOOL;
	Name		: Core.T_MaxString;
	Axis		: REFERENCE TO AXIS_REF;
END_VAR
// Register all Motion Tasks to Collection
MotionTaskCollection.AddTask(MoveAbsoluteTask);
MotionTaskCollection.AddTask(MoveRelativeTask);
MotionTaskCollection.AddTask(MoveModuloTask);
MotionTaskCollection.AddTask(MoveVelocityTask);
END_METHOD

METHOD MoveAbsolute
VAR_INPUT
	TargetPosition : LREAL;
	AbortPrevious  : BOOL := TRUE;
END_VAR
IF Error THEN
	RETURN;
ELSE
	IF Busy AND NOT AbortPrevious THEN
		RETURN;
	END_IF
END_IF

MoveAbsoluteTask.BufferMode		:= _McBufferMode;
MoveAbsoluteTask.MoveOptions	:= _MoveOptions;
MoveAbsoluteTask.TargetPosition := TargetPosition;
MoveAbsoluteTask.Execute();
END_METHOD

METHOD MoveModulo : BOOL
VAR_INPUT
	Position	: LREAL;
	Direction	: MC_Direction := .MC_Direction.MC_Shortest_Way;
	AbortPrevious	: BOOL := TRUE;
END_VAR
IF Error THEN
	RETURN;
ELSE
	IF Busy AND NOT AbortPrevious THEN
		RETURN;
	END_IF
END_IF

MoveModuloTask.BufferMode	  := _McBufferMode;
MoveModuloTask.MoveOptions	  := _MoveOptions;
MoveModuloTask.Direction	  := Direction;
MoveModuloTask.TargetPosition := Position;
MoveModuloTask.Execute();
END_METHOD

METHOD MoveRelative : BOOL
VAR_INPUT
	Distance	  : LREAL;
	AbortPrevious : BOOL := TRUE;
END_VAR
IF Error THEN
	RETURN;
ELSE
	IF Busy AND NOT AbortPrevious THEN
		RETURN;
	END_IF
END_IF

MoveRelativeTask.BufferMode		:= _McBufferMode;
MoveRelativeTask.MoveOptions	:= _MoveOptions;
MoveRelativeTask.TargetDistance := Distance;
MoveRelativeTask.Execute();
END_METHOD

METHOD MoveVelocity : BOOL
VAR_INPUT
	Velocity	  : LREAL;
	AbortPrevious : BOOL := TRUE;
END_VAR
IF Error THEN
	RETURN;
ELSE
	IF Busy AND NOT AbortPrevious THEN
		RETURN;
	END_IF
END_IF

MoveVelocityTask.BufferMode		:= _McBufferMode;
MoveVelocityTask.MoveOptions	:= _MoveOptions;
MoveVelocityTask.TargetVelocity := Velocity;
MoveVelocityTask.Execute();
END_METHOD

END_FUNCTION_BLOCK

// Motion/AxisPTP_HMI
FUNCTION_BLOCK AxisPTP_HMI EXTENDS HmiFunction
VAR
	Axis : I_Axis_PTP;
	{ attribute 'TcHmiSymbol.AddSymbol' }
	{ attribute 'TcHmiSymbol.AddSymbol.UserGroups' := '__SystemAdministrators,Admin' }
	AxisPTP_HMI : ST_AxisPTP_HMI;
END_VAR

PROPERTY DisablePermissive : I_Permissive
GET
DisablePermissive := AxisPTP_HMI.Disable.Permissive;
END_GET
END_PROPERTY

PROPERTY EnablePermissive : I_Permissive
GET
EnablePermissive := AxisPTP_HMI.Enable.Permissive;
END_GET
END_PROPERTY

PROPERTY HomePermissive : I_Permissive
GET
HomePermissive := AxisPTP_HMI.Home.Permissive;
END_GET
END_PROPERTY

PROPERTY JogBackwardFastPermissive : I_Permissive
GET
JogBackwardFastPermissive := AxisPTP_HMI.JogBackwardFast.Permissive;
END_GET
END_PROPERTY

PROPERTY JogBackwardSlowPermissive : I_Permissive
GET
JogBackwardSlowPermissive := AxisPTP_HMI.JogBackwardSlow.Permissive;
END_GET
END_PROPERTY

PROPERTY JogForwardFastPermissive : I_Permissive
GET
JogForwardFastPermissive := AxisPTP_HMI.JogForwardFast.Permissive;
END_GET
END_PROPERTY

PROPERTY JogForwardSlowPermissive : I_Permissive
GET
JogForwardSlowPermissive := AxisPTP_HMI.JogForwardSlow.Permissive;
END_GET
END_PROPERTY

PROPERTY MoveAbsolutePermissive : I_Permissive
GET
MoveAbsolutePermissive := AxisPTP_HMI.MoveAbsolute.Permissive;
END_GET
END_PROPERTY

PROPERTY MoveModuloPermissive : I_Permissive
GET
MoveModuloPermissive := AxisPTP_HMI.MoveModulo.Permissive;
END_GET
END_PROPERTY

PROPERTY MoveRelativePermissive : I_Permissive
GET
MoveRelativePermissive := AxisPTP_HMI.MoveRelative.Permissive;
END_GET
END_PROPERTY

PROPERTY MoveVelocityPermissive : I_Permissive
GET
MoveVelocityPermissive := AxisPTP_HMI.MoveVelocity.Permissive;
END_GET
END_PROPERTY

PROPERTY ResetPermissive : I_Permissive
GET
ResetPermissive := AxisPTP_HMI.Reset.Permissive;
END_GET
END_PROPERTY

PROPERTY StopPermissive : I_Permissive
GET
StopPermissive := AxisPTP_HMI.Stop.Permissive;
END_GET
END_PROPERTY

PROPERTY ControlObject : I_Base
SET
__QueryInterface(ControlObject,Axis);
END_SET
END_PROPERTY

METHOD CyclicLogic
VAR_INST
	EnableRT	   : R_TRIG;
	DisableRT	   : R_TRIG;
	StopRT		   : R_TRIG;
	HomeRT		   : R_TRIG;
	ResetRT		   : R_TRIG;
	MoveAbsoluteRT : R_TRIG;
	MoveModuloRT   : R_TRIG;
	MoveRelativeRT : R_TRIG;
	MoveVelocityRT : R_TRIG;
END_VAR
IF Axis = 0 THEN
	RETURN;
END_IF

AxisPTP_HMI.HmiEnabled			 := Enabled;
AxisPTP_HMI.ActualAcceleration	 := Axis.ActualAcceleration;
AxisPTP_HMI.ActualPosition		 := Axis.ActualPosition;
AxisPTP_HMI.ActualPositionModulo := Axis.ActualPositionModulo;
AxisPTP_HMI.ActualTorque		 := Axis.ActualTorque;
AxisPTP_HMI.ActualVelocity		 := Axis.ActualVelocity;
AxisPTP_HMI.Busy				 := Axis.Busy;
AxisPTP_HMI.Error				 := Axis.Error;
AxisPTP_HMI.ErrorId				 := Axis.ErrorId;
AxisPTP_HMI.Name				 := Axis.Name;
AxisPTP_HMI.Status				 := Axis.Axis.Status;

// HMI Commands
StopRT(CLK := AxisPTP_HMI.Stop.Active);
IF StopRT.Q THEN
	IF AxisPTP_HMI.Stop.Permissive.OK THEN
		Axis.Stop();
	END_IF
END_IF

ResetRT(CLK := AxisPTP_HMI.Reset.Active);
IF ResetRT.Q THEN
	IF AxisPTP_HMI.Reset.Permissive.OK THEN
		Axis.Reset();
	END_IF
END_IF

IF Enabled THEN
	EnableRT(CLK := AxisPTP_HMI.Enable.Active);
	IF EnableRT.Q THEN
		IF AxisPTP_HMI.Enable.Permissive.OK THEN
			Axis.Enable();
		END_IF
	END_IF

	DisableRT(CLK := AxisPTP_HMI.Disable.Active);
	IF DisableRT.Q THEN
		IF AxisPTP_HMI.Disable.Permissive.OK THEN
			Axis.Disable();
		END_IF
	END_IF

	IF AxisPTP_HMI.JogBackwardSlow.Active THEN
		IF AxisPTP_HMI.JogBackwardSlow.Permissive.OK THEN
			Axis.Jog(JogForward := FALSE, JogBackwards := TRUE, JogMode := E_JogMode.MC_JOGMODE_STANDARD_SLOW);
		END_IF
	ELSIF AxisPTP_HMI.JogForwardSlow.Active THEN
		Axis.Jog(JogForward := TRUE, JogBackwards := FALSE, JogMode := E_JogMode.MC_JOGMODE_STANDARD_SLOW);
	ELSIF AxisPTP_HMI.JogBackwardFast.Active THEN
		Axis.Jog(JogForward := FALSE, JogBackwards := TRUE, JogMode := E_JogMode.MC_JOGMODE_STANDARD_FAST);
	ELSIF AxisPTP_HMI.JogForwardFast.Active THEN
		Axis.Jog(JogForward := TRUE, JogBackwards := FALSE, JogMode := E_JogMode.MC_JOGMODE_STANDARD_FAST);
	ELSE
		Axis.Jog(JogForward := FALSE, JogBackwards := FALSE, JogMode := E_JogMode.MC_JOGMODE_STANDARD_SLOW);
	END_IF

	HomeRT(CLK := AxisPTP_HMI.Home.Active);
	IF HomeRT.Q THEN
		IF AxisPTP_HMI.Home.Permissive.OK THEN
			Axis.Home();
		END_IF
	END_IF

	MoveAbsoluteRT(CLK := AxisPTP_HMI.MoveAbsolute.Active);
	IF MoveAbsoluteRT.Q THEN
		IF AxisPTP_HMI.MoveAbsolute.Permissive.OK THEN
			Axis.MoveAbsolute(AxisPTP_HMI.TargetPosition);
		END_IF
	END_IF

	MoveModuloRT(CLK := AxisPTP_HMI.MoveModulo.Active);
	IF MoveModuloRT.Q THEN
		IF AxisPTP_HMI.MoveModulo.Permissive.OK THEN
			Axis.MoveModulo(AxisPTP_HMI.TargetPosition);
		END_IF
	END_IF

	MoveRelativeRT(CLK := AxisPTP_HMI.MoveRelative.Active);
	IF MoveRelativeRT.Q THEN
		IF AxisPTP_HMI.MoveRelative.Permissive.OK THEN
			Axis.MoveRelative(AxisPTP_HMI.TargetDistance);
		END_IF
	END_IF

	MoveVelocityRT(CLK := AxisPTP_HMI.MoveVelocity.Active);
	IF MoveVelocityRT.Q THEN
		IF AxisPTP_HMI.MoveVelocity.Permissive.OK THEN
			Axis.MoveVelocity(AxisPTP_HMI.TargetVelocity);
		END_IF
	END_IF
END_IF
END_METHOD

(*FB_Init is always available implicitly and it is used primarily for initialization.
The return value is not evaluated. For a specific influence, you can also declare the
methods explicitly and provide additional code there with the standard initialization
code. You can evaluate the return value.*)
METHOD FB_Init : BOOL
VAR_INPUT
	(* TRUE: the retain variables are initialized (reset warm / reset cold)*)
	bInitRetains : BOOL;

	(* TRUE: the instance will be copied to the copy code afterward (online change)   *)
	bInCopyCode : BOOL;
	Name		: Core.T_MaxString;
	Axis		: I_Axis_PTP;
	Unit		: STRING;
END_VAR
THIS^.Axis		 := Axis;
ControlType		 := 'AxisPTP';
LinkObject		 := 'AxisPTP_HMI';
AxisPTP_HMI.Unit := Unit;
END_METHOD

END_FUNCTION_BLOCK

// Motion/SlaveAxisPTP
FUNCTION_BLOCK SlaveAxisPTP EXTENDS AxisPTP IMPLEMENTS I_SlaveAxis
VAR
	// Tasks
	MotionCoupleTaskGearing : MotionCoupleTask_Gearing := (Name := 'MC GearIn Multimaster');
END_VAR

(*FB_Init is always available implicitly and it is used primarily for initialization.
The return value is not evaluated. For a specific influence, you can also declare the
methods explicitly and provide additional code there with the standard initialization
code. You can evaluate the return value.*)
METHOD FB_Init : BOOL
VAR_INPUT
	(* TRUE: the retain variables are initialized (reset warm / reset cold)*)
	bInitRetains : BOOL;

	(* TRUE: the instance will be copied to the copy code afterward (online change)   *)
	bInCopyCode : BOOL;
	Name		: Core.T_MaxString;
	Axis		: REFERENCE TO AXIS_REF;
END_VAR
// Register all Motion Tasks to Collection
MotionTaskCollection.AddTask(MotionCoupleTaskGearing);
END_METHOD

METHOD GearIn
VAR_INPUT
END_VAR
MotionCoupleTaskGearing.GearIn	   := TRUE;
MotionCoupleTaskGearing.BufferMode := _McBufferMode;
MotionCoupleTaskGearing.Execute();
END_METHOD

PROPERTY GearInMultiMasterOptions : ST_GearInMultiMasterOptions
SET
MotionCoupleTaskGearing.GearInMultiMasterOptions := GearInMultiMasterOptions;
END_SET
END_PROPERTY

METHOD GearOut
VAR_INPUT
END_VAR
MotionCoupleTaskGearing.GearIn := FALSE;
MotionCoupleTaskGearing.Execute();
END_METHOD

{attribute 'monitoring' := 'call'}
PROPERTY GearRatioMaster1 : LREAL
SET
MotionCoupleTaskGearing.GearRatioMaster1 := GearRatioMaster1;
END_SET
END_PROPERTY

{attribute 'monitoring' := 'call'}
PROPERTY GearRatioMaster2 : LREAL
SET
MotionCoupleTaskGearing.GearRatioMaster2 := GearRatioMaster2;
END_SET
END_PROPERTY

{attribute 'monitoring' := 'call'}
PROPERTY GearRatioMaster3 : LREAL
SET
MotionCoupleTaskGearing.GearRatioMaster3 := GearRatioMaster3;
END_SET
END_PROPERTY

{attribute 'monitoring' := 'call'}
PROPERTY GearRatioMaster4 : LREAL
SET
MotionCoupleTaskGearing.GearRatioMaster4 := GearRatioMaster4;
END_SET
END_PROPERTY

PROPERTY Master1 : I_Axis
SET
MotionCoupleTaskGearing.Master1 := Master1;
END_SET
END_PROPERTY

PROPERTY Master2 : I_Axis
SET
MotionCoupleTaskGearing.Master2 := Master2;
END_SET
END_PROPERTY

PROPERTY Master3 : I_Axis
SET
MotionCoupleTaskGearing.Master3 := Master3;
END_SET
END_PROPERTY

PROPERTY Master4 : I_Axis
SET
MotionCoupleTaskGearing.Master4 := Master4;
END_SET
END_PROPERTY

END_FUNCTION_BLOCK

// Project Information/F_GetCompany
// This function has been automatically generated from the project information.
{attribute 'signature_flag' := '1073741824'}
{attribute 'TcGenerated'}
{attribute 'no-analysis'}
FUNCTION F_GetCompany : WSTRING
VAR_INPUT
	
END_VAR

F_GetCompany := "Beckhoff Automation LLC";

END_FUNCTION

// Project Information/F_GetTitle
// This function has been automatically generated from the project information.
{attribute 'signature_flag' := '1073741824'}
{attribute 'TcGenerated'}
{attribute 'no-analysis'}
FUNCTION F_GetTitle : WSTRING
VAR_INPUT
	
END_VAR

F_GetTitle := "CoreMotionNc2";

END_FUNCTION

// Project Information/F_GetVersion
// This function has been automatically generated from the project information.
{attribute 'signature_flag' := '1073741824'}
{attribute 'TcGenerated'}
{attribute 'no-analysis'}
FUNCTION F_GetVersion : ST_LibVersion
VAR_INPUT
	
END_VAR

F_GetVersion.iMajor := 1;
F_GetVersion.iMinor := 1;
F_GetVersion.iBuild := 8;
F_GetVersion.iRevision := 0;
F_GetVersion.sVersion := '1.1.8';
F_GetVersion.nFlags := 0;

END_FUNCTION
